    |   movel([0.087836, -1.394012, -2.564950, -0.753428, 1.570796, 1.658633],accel_mss,speed_ms,0,blend_radius_m)
    |   movel([0.088216, -1.393731, -2.565153, -0.753505, 1.570796, 1.659012],accel_mss,speed_ms,0,blend_radius_m)
    |   movel([0.088598, -1.393563, -2.565275, -0.753551, 1.570796, 1.659394],accel_mss,speed_ms,0,blend_radius_m)
    |   movel([0.088951, -1.393516, -2.565308, -0.753564, 1.570796, 1.659747],accel_mss,speed_ms,0,blend_radius_m)
    |   movel([0.089293, -1.393576, -2.565265, -0.753548, 1.570796, 1.660089],accel_mss,speed_ms,0,blend_radius_m)
    |   speed_ms = 0.003
    |   movel([0.089293, -1.380644, -2.559336, -0.772409, 1.570796, 1.660089],accel_mss,speed_ms,0,blend_radius_m)
    |   speed_ms = 1.000
    |   movel([0.089293, -1.355826, -2.547083, -0.809480, 1.570796, 1.660089],accel_mss,speed_ms,0,blend_radius_m)
    |   movel([0.088410, -1.349799, -2.551181, -0.811409, 1.570796, 1.659206],accel_mss,speed_ms,0,blend_radius_m)
    |   movel([0.088410, -1.374726, -2.563511, -0.774153, 1.570796, 1.659206],accel_mss,speed_ms,0,blend_radius_m)
    |   speed_ms = 0.003
    |   movel([0.088410, -1.384438, -2.567999, -0.759952, 1.570796, 1.659206],accel_mss,speed_ms,0,blend_radius_m)
    |   speed_ms = 0.007
    |   movel([0.087081, -1.384926, -2.567651, -0.759811, 1.570796, 1.657878],accel_mss,speed_ms,0,blend_radius_m)
    |   movel([0.085949, -1.385546, -2.567210, -0.759633, 1.570796, 1.656745],accel_mss,speed_ms,0,blend_radius_m)
    |   movel([0.084872, -1.386318, -2.566658, -0.759412, 1.570796, 1.655668],accel_mss,speed_ms,0,blend_radius_m)
    |   movel([0.083929, -1.387193, -2.566033, -0.759163, 1.570796, 1.654725],accel_mss,speed_ms,0,blend_radius_m)
    |   movel([0.083360, -1.387850, -2.565563, -0.758976, 1.570796, 1.654157],accel_mss,speed_ms,0,blend_radius_m)
    |   movel([0.082732, -1.388688, -2.564962, -0.758739, 1.570796, 1.653528],accel_mss,speed_ms,0,blend_radius_m)
    |   movel([0.082181, -1.389503, -2.564376, -0.758510, 1.570796, 1.652978],accel_mss,speed_ms,0,blend_radius_m)
    |   movel([0.081904, -1.390039, -2.563990, -0.758359, 1.570796, 1.652700],accel_mss,speed_ms,0,blend_radius_m)
    |   movel([0.081705, -1.390252, -2.563838, -0.758300, 1.570796, 1.652502],accel_mss,speed_ms,0,blend_radius_m)
    |   movel([0.081566, -1.390049, -2.563984, -0.758357, 1.570796, 1.652362],accel_mss,speed_ms,0,blend_radius_m)
    |   movel([0.081299, -1.389034, -2.564713, -0.758642, 1.570796, 1.652095],accel_mss,speed_ms,0,blend_radius_m)
    |   movel([0.081058, -1.387988, -2.565464, -0.758937, 1.570796, 1.651854],accel_mss,speed_ms,0,blend_radius_m)
    |   movel([0.080915, -1.387123, -2.566083, -0.759183, 1.570796, 1.651712],accel_mss,speed_ms,0,blend_radius_m)
    |   movel([0.080836, -1.386274, -2.566690, -0.759425, 1.570796, 1.651632],accel_mss,speed_ms,0,blend_radius_m)
    |   movel([0.080928, -1.385938, -2.566930, -0.759521, 1.570796, 1.651725],accel_mss,speed_ms,0,blend_radius_m)
    |   movel([0.081186, -1.385742, -2.567070, -0.759577, 1.570796, 1.651983],accel_mss,speed_ms,0,blend_radius_m)
    |   movel([0.081800, -1.385622, -2.567155, -0.759611, 1.570796, 1.652596],accel_mss,speed_ms,0,blend_radius_m)
    |   movel([0.082664, -1.385488, -2.567251, -0.759650, 1.570796, 1.653461],accel_mss,speed_ms,0,blend_radius_m)
    |   movel([0.083900, -1.385238, -2.567429, -0.759721, 1.570796, 1.654697],accel_mss,speed_ms,0,blend_radius_m)
    |   movel([0.085342, -1.384916, -2.567659, -0.759814, 1.570796, 1.656138],accel_mss,speed_ms,0,blend_radius_m)
    |   movel([0.086879, -1.384542, -2.567925, -0.759922, 1.570796, 1.657675],accel_mss,speed_ms,0,blend_radius_m)
    |   movel([0.087796, -1.384317, -2.568085, -0.759987, 1.570796, 1.658593],accel_mss,speed_ms,0,blend_radius_m)
    |   movel([0.088317, -1.384208, -2.568162, -0.760018, 1.570796, 1.659114],accel_mss,speed_ms,0,blend_radius_m)
    |   movel([0.088631, -1.384168, -2.568191, -0.760030, 1.570796, 1.659427],accel_mss,speed_ms,0,blend_radius_m)
    |   movel([0.088410, -1.384438, -2.567999, -0.759952, 1.570796, 1.659206],accel_mss,speed_ms,0,blend_radius_m)
    |   speed_ms = 0.003
    |   movel([0.088410, -1.387720, -2.569479, -0.755191, 1.570796, 1.659206],accel_mss,speed_ms,0,blend_radius_m)
    |   speed_ms = 0.007
    |   movel([0.087081, -1.388207, -2.569130, -0.755052, 1.570796, 1.657878],accel_mss,speed_ms,0,blend_radius_m)
    |   movel([0.085949, -1.388825, -2.568687, -0.754877, 1.570796, 1.656745],accel_mss,speed_ms,0,blend_radius_m)
    |   movel([0.084872, -1.389595, -2.568135, -0.754659, 1.570796, 1.655668],accel_mss,speed_ms,0,blend_radius_m)
    |   movel([0.083929, -1.390467, -2.567508, -0.754414, 1.570796, 1.654725],accel_mss,speed_ms,0,blend_radius_m)
    |   movel([0.083360, -1.391123, -2.567036, -0.754230, 1.570796, 1.654157],accel_mss,speed_ms,0,blend_radius_m)
    |   movel([0.082732, -1.391958, -2.566434, -0.753997, 1.570796, 1.653528],accel_mss,speed_ms,0,blend_radius_m)
    |   movel([0.082181, -1.392771, -2.565848, -0.753771, 1.570796, 1.652978],accel_mss,speed_ms,0,blend_radius_m)
    |   movel([0.081904, -1.393306, -2.565461, -0.753622, 1.570796, 1.652700],accel_mss,speed_ms,0,blend_radius_m)
    |   movel([0.081705, -1.393518, -2.565308, -0.753564, 1.570796, 1.652502],accel_mss,speed_ms,0,blend_radius_m)
    |   movel([0.081566, -1.393315, -2.565454, -0.753620, 1.570796, 1.652362],accel_mss,speed_ms,0,blend_radius_m)
    |   movel([0.081299, -1.392304, -2.566185, -0.753900, 1.570796, 1.652095],accel_mss,speed_ms,0,blend_radius_m)
    |   movel([0.081058, -1.391260, -2.566937, -0.754191, 1.570796, 1.651854],accel_mss,speed_ms,0,blend_radius_m)
    |   movel([0.080915, -1.390398, -2.567558, -0.754433, 1.570796, 1.651712],accel_mss,speed_ms,0,blend_radius_m)
    |   movel([0.080836, -1.389551, -2.568167, -0.754672, 1.570796, 1.651632],accel_mss,speed_ms,0,blend_radius_m)
    |   movel([0.080928, -1.389216, -2.568407, -0.754766, 1.570796, 1.651725],accel_mss,speed_ms,0,blend_radius_m)
    |   movel([0.081186, -1.389020, -2.568547, -0.754822, 1.570796, 1.651983],accel_mss,speed_ms,0,blend_radius_m)
    |   movel([0.081800, -1.388901, -2.568633, -0.754855, 1.570796, 1.652596],accel_mss,speed_ms,0,blend_radius_m)
    |   movel([0.082664, -1.388767, -2.568728, -0.754893, 1.570796, 1.653461],accel_mss,speed_ms,0,blend_radius_m)
    |   movel([0.083900, -1.388518, -2.568907, -0.754964, 1.570796, 1.654697],accel_mss,speed_ms,0,blend_radius_m)
    |   movel([0.085342, -1.388196, -2.569138, -0.755055, 1.570796, 1.656138],accel_mss,speed_ms,0,blend_radius_m)
    |   movel([0.086879, -1.387824, -2.569404, -0.755161, 1.570796, 1.657675],accel_mss,speed_ms,0,blend_radius_m)
    |   movel([0.087796, -1.387599, -2.569565, -0.755225, 1.570796, 1.658593],accel_mss,speed_ms,0,blend_radius_m)
    |   movel([0.088317, -1.387491, -2.569642, -0.755256, 1.570796, 1.659114],accel_mss,speed_ms,0,blend_radius_m)
    |   movel([0.088631, -1.387451, -2.569671, -0.755267, 1.570796, 1.659427],accel_mss,speed_ms,0,blend_radius_m)
    |   movel([0.088410, -1.387720, -2.569479, -0.755191, 1.570796, 1.659206],accel_mss,speed_ms,0,blend_radius_m)
    |   speed_ms = 0.003
    |   movel([0.088410, -1.374726, -2.563511, -0.774153, 1.570796, 1.659206],accel_mss,speed_ms,0,blend_radius_m)
    |   speed_ms = 1.000
    |   movel([0.088410, -1.349799, -2.551181, -0.811409, 1.570796, 1.659206],accel_mss,speed_ms,0,blend_radius_m)
    |   movel([0.072038, -1.358116, -2.545513, -0.808760, 1.570796, 1.642834],accel_mss,speed_ms,0,blend_radius_m)
    |   movel([0.072038, -1.382893, -2.557737, -0.771760, 1.570796, 1.642834],accel_mss,speed_ms,0,blend_radius_m)
    |   speed_ms = 0.003
    |   movel([0.072038, -1.392541, -2.562186, -0.757663, 1.570796, 1.642834],accel_mss,speed_ms,0,blend_radius_m)
    |   speed_ms = 0.007
    |   movel([0.072079, -1.392738, -2.562043, -0.757608, 1.570796, 1.642875],accel_mss,speed_ms,0,blend_radius_m)
    |   movel([0.071854, -1.393010, -2.561846, -0.757533, 1.570796, 1.642650],accel_mss,speed_ms,0,blend_radius_m)
    |   movel([0.071545, -1.393082, -2.561794, -0.757513, 1.570796, 1.642341],accel_mss,speed_ms,0,blend_radius_m)
    |   movel([0.071303, -1.393090, -2.561788, -0.757511, 1.570796, 1.642100],accel_mss,speed_ms,0,blend_radius_m)
    |   movel([0.071035, -1.393108, -2.561775, -0.757506, 1.570796, 1.641831],accel_mss,speed_ms,0,blend_radius_m)
    |   movel([0.070605, -1.393174, -2.561727, -0.757488, 1.570796, 1.641402],accel_mss,speed_ms,0,blend_radius_m)
    |   movel([0.070116, -1.393271, -2.561657, -0.757461, 1.570796, 1.640912],accel_mss,speed_ms,0,blend_radius_m)
    |   movel([0.069632, -1.393385, -2.561575, -0.757430, 1.570796, 1.640429],accel_mss,speed_ms,0,blend_radius_m)
    |   movel([0.068674, -1.393599, -2.561419, -0.757371, 1.570796, 1.639470],accel_mss,speed_ms,0,blend_radius_m)
    |   movel([0.068254, -1.393580, -2.561433, -0.757376, 1.570796, 1.639050],accel_mss,speed_ms,0,blend_radius_m)
    |   movel([0.068198, -1.393373, -2.561583, -0.757433, 1.570796, 1.638995],accel_mss,speed_ms,0,blend_radius_m)
    |   movel([0.068476, -1.392973, -2.561872, -0.757543, 1.570796, 1.639272],accel_mss,speed_ms,0,blend_radius_m)
    |   movel([0.068846, -1.392690, -2.562077, -0.757621, 1.570796, 1.639642],accel_mss,speed_ms,0,blend_radius_m)
    |   movel([0.069096, -1.392605, -2.562139, -0.757645, 1.570796, 1.639893],accel_mss,speed_ms,0,blend_radius_m)
    |   movel([0.069570, -1.392494, -2.562220, -0.757676, 1.570796, 1.640367],accel_mss,speed_ms,0,blend_radius_m)
    |   movel([0.070403, -1.392329, -2.562339, -0.757721, 1.570796, 1.641200],accel_mss,speed_ms,0,blend_radius_m)
    |   movel([0.071125, -1.392221, -2.562417, -0.757751, 1.570796, 1.641922],accel_mss,speed_ms,0,blend_radius_m)
    |   movel([0.071701, -1.392164, -2.562458, -0.757767, 1.570796, 1.642497],accel_mss,speed_ms,0,blend_radius_m)
    |   movel([0.071942, -1.392284, -2.562371, -0.757734, 1.570796, 1.642738],accel_mss,speed_ms,0,blend_radius_m)
    |   movel([0.072038, -1.392541, -2.562186, -0.757663, 1.570796, 1.642834],accel_mss,speed_ms,0,blend_radius_m)
    |   speed_ms = 0.003
    |   movel([0.072038, -1.395800, -2.563652, -0.752937, 1.570796, 1.642834],accel_mss,speed_ms,0,blend_radius_m)
    |   speed_ms = 0.007
    |   movel([0.072079, -1.395997, -2.563509, -0.752883, 1.570796, 1.642875],accel_mss,speed_ms,0,blend_radius_m)
    |   movel([0.071854, -1.396269, -2.563311, -0.752809, 1.570796, 1.642650],accel_mss,speed_ms,0,blend_radius_m)
    |   movel([0.071545, -1.396340, -2.563259, -0.752790, 1.570796, 1.642341],accel_mss,speed_ms,0,blend_radius_m)
    |   movel([0.071303, -1.396348, -2.563254, -0.752788, 1.570796, 1.642100],accel_mss,speed_ms,0,blend_radius_m)
    |   movel([0.071035, -1.396366, -2.563240, -0.752783, 1.570796, 1.641831],accel_mss,speed_ms,0,blend_radius_m)
    |   movel([0.070605, -1.396432, -2.563192, -0.752765, 1.570796, 1.641402],accel_mss,speed_ms,0,blend_radius_m)
    |   movel([0.070116, -1.396529, -2.563122, -0.752738, 1.570796, 1.640912],accel_mss,speed_ms,0,blend_radius_m)
    |   movel([0.069632, -1.396642, -2.563039, -0.752708, 1.570796, 1.640429],accel_mss,speed_ms,0,blend_radius_m)
    |   movel([0.068674, -1.396856, -2.562883, -0.752649, 1.570796, 1.639470],accel_mss,speed_ms,0,blend_radius_m)
    |   movel([0.068254, -1.396836, -2.562898, -0.752655, 1.570796, 1.639050],accel_mss,speed_ms,0,blend_radius_m)
    |   movel([0.068198, -1.396630, -2.563048, -0.752711, 1.570796, 1.638995],accel_mss,speed_ms,0,blend_radius_m)
    |   movel([0.068476, -1.396232, -2.563338, -0.752819, 1.570796, 1.639272],accel_mss,speed_ms,0,blend_radius_m)
    |   movel([0.068846, -1.395949, -2.563543, -0.752896, 1.570796, 1.639642],accel_mss,speed_ms,0,blend_radius_m)
    |   movel([0.069096, -1.395864, -2.563605, -0.752919, 1.570796, 1.639893],accel_mss,speed_ms,0,blend_radius_m)
    |   movel([0.069570, -1.395754, -2.563686, -0.752950, 1.570796, 1.640367],accel_mss,speed_ms,0,blend_radius_m)
    |   movel([0.070403, -1.395589, -2.563805, -0.752995, 1.570796, 1.641200],accel_mss,speed_ms,0,blend_radius_m)
    |   movel([0.071125, -1.395481, -2.563884, -0.753024, 1.570796, 1.641922],accel_mss,speed_ms,0,blend_radius_m)
    |   movel([0.071701, -1.395425, -2.563925, -0.753040, 1.570796, 1.642497],accel_mss,speed_ms,0,blend_radius_m)
    |   movel([0.071942, -1.395544, -2.563838, -0.753007, 1.570796, 1.642738],accel_mss,speed_ms,0,blend_radius_m)
    |   movel([0.072038, -1.395800, -2.563652, -0.752937, 1.570796, 1.642834],accel_mss,speed_ms,0,blend_radius_m)
    |   speed_ms = 0.003
    |   movel([0.072038, -1.382893, -2.557737, -0.771760, 1.570796, 1.642834],accel_mss,speed_ms,0,blend_radius_m)
    |   speed_ms = 1.000
    |   movel([0.072038, -1.358116, -2.545513, -0.808760, 1.570796, 1.642834],accel_mss,speed_ms,0,blend_radius_m)
    |   movel([0.071087, -1.359327, -2.544680, -0.808382, 1.570796, 1.641883],accel_mss,speed_ms,0,blend_radius_m)
    |   movel([0.071087, -1.384082, -2.556888, -0.771419, 1.570796, 1.641883],accel_mss,speed_ms,0,blend_radius_m)
    |   speed_ms = 0.003
    |   movel([0.071087, -1.393720, -2.561331, -0.757337, 1.570796, 1.641883],accel_mss,speed_ms,0,blend_radius_m)
    |   speed_ms = 0.007
    |   movel([0.071759, -1.393816, -2.561262, -0.757311, 1.570796, 1.642556],accel_mss,speed_ms,0,blend_radius_m)
    |   movel([0.071953, -1.393945, -2.561168, -0.757276, 1.570796, 1.642749],accel_mss,speed_ms,0,blend_radius_m)
    |   movel([0.072032, -1.394114, -2.561046, -0.757229, 1.570796, 1.642829],accel_mss,speed_ms,0,blend_radius_m)
    |   movel([0.071840, -1.394423, -2.560821, -0.757144, 1.570796, 1.642637],accel_mss,speed_ms,0,blend_radius_m)
    |   movel([0.071514, -1.394499, -2.560766, -0.757124, 1.570796, 1.642311],accel_mss,speed_ms,0,blend_radius_m)
    |   movel([0.071242, -1.394533, -2.560742, -0.757114, 1.570796, 1.642039],accel_mss,speed_ms,0,blend_radius_m)
    |   movel([0.070950, -1.394556, -2.560725, -0.757108, 1.570796, 1.641746],accel_mss,speed_ms,0,blend_radius_m)
    |   movel([0.070596, -1.394590, -2.560700, -0.757099, 1.570796, 1.641393],accel_mss,speed_ms,0,blend_radius_m)
    |   movel([0.070127, -1.394658, -2.560651, -0.757080, 1.570796, 1.640923],accel_mss,speed_ms,0,blend_radius_m)
    |   movel([0.069629, -1.394746, -2.560587, -0.757056, 1.570796, 1.640426],accel_mss,speed_ms,0,blend_radius_m)
    |   movel([0.069177, -1.394842, -2.560517, -0.757030, 1.570796, 1.639973],accel_mss,speed_ms,0,blend_radius_m)
    |   movel([0.068658, -1.394956, -2.560434, -0.756999, 1.570796, 1.639454],accel_mss,speed_ms,0,blend_radius_m)
    |   movel([0.068335, -1.395002, -2.560401, -0.756986, 1.570796, 1.639131],accel_mss,speed_ms,0,blend_radius_m)
    |   movel([0.068017, -1.394943, -2.560443, -0.757002, 1.570796, 1.638813],accel_mss,speed_ms,0,blend_radius_m)
    |   movel([0.068021, -1.394682, -2.560633, -0.757074, 1.570796, 1.638818],accel_mss,speed_ms,0,blend_radius_m)
    |   movel([0.068685, -1.394201, -2.560983, -0.757205, 1.570796, 1.639482],accel_mss,speed_ms,0,blend_radius_m)
    |   movel([0.069886, -1.393897, -2.561203, -0.757289, 1.570796, 1.640683],accel_mss,speed_ms,0,blend_radius_m)
    |   movel([0.071087, -1.393720, -2.561331, -0.757337, 1.570796, 1.641883],accel_mss,speed_ms,0,blend_radius_m)
    |   speed_ms = 0.003
    |   movel([0.071087, -1.396977, -2.562796, -0.752617, 1.570796, 1.641883],accel_mss,speed_ms,0,blend_radius_m)
    |   speed_ms = 0.007
    |   movel([0.071759, -1.397072, -2.562726, -0.752591, 1.570796, 1.642556],accel_mss,speed_ms,0,blend_radius_m)
    |   movel([0.071953, -1.397201, -2.562632, -0.752556, 1.570796, 1.642749],accel_mss,speed_ms,0,blend_radius_m)
    |   movel([0.072032, -1.397369, -2.562509, -0.752510, 1.570796, 1.642829],accel_mss,speed_ms,0,blend_radius_m)
    |   movel([0.071840, -1.397678, -2.562284, -0.752427, 1.570796, 1.642637],accel_mss,speed_ms,0,blend_radius_m)
    |   movel([0.071514, -1.397753, -2.562229, -0.752406, 1.570796, 1.642311],accel_mss,speed_ms,0,blend_radius_m)
    |   movel([0.071242, -1.397787, -2.562205, -0.752397, 1.570796, 1.642039],accel_mss,speed_ms,0,blend_radius_m)
    |   movel([0.070950, -1.397810, -2.562188, -0.752391, 1.570796, 1.641746],accel_mss,speed_ms,0,blend_radius_m)
    |   movel([0.070596, -1.397844, -2.562163, -0.752382, 1.570796, 1.641393],accel_mss,speed_ms,0,blend_radius_m)
    |   movel([0.070127, -1.397911, -2.562114, -0.752364, 1.570796, 1.640923],accel_mss,speed_ms,0,blend_radius_m)
    |   movel([0.069629, -1.398000, -2.562049, -0.752340, 1.570796, 1.640426],accel_mss,speed_ms,0,blend_radius_m)
    |   movel([0.069177, -1.398096, -2.561979, -0.752314, 1.570796, 1.639973],accel_mss,speed_ms,0,blend_radius_m)
    |   movel([0.068658, -1.398209, -2.561896, -0.752283, 1.570796, 1.639454],accel_mss,speed_ms,0,blend_radius_m)
    |   movel([0.068335, -1.398255, -2.561863, -0.752271, 1.570796, 1.639131],accel_mss,speed_ms,0,blend_radius_m)
    |   movel([0.068017, -1.398196, -2.561906, -0.752287, 1.570796, 1.638813],accel_mss,speed_ms,0,blend_radius_m)
    |   movel([0.068021, -1.397936, -2.562096, -0.752357, 1.570796, 1.638818],accel_mss,speed_ms,0,blend_radius_m)
    |   movel([0.068685, -1.397456, -2.562446, -0.752487, 1.570796, 1.639482],accel_mss,speed_ms,0,blend_radius_m)
    |   movel([0.069886, -1.397153, -2.562667, -0.752569, 1.570796, 1.640683],accel_mss,speed_ms,0,blend_radius_m)
    |   movel([0.071087, -1.396977, -2.562796, -0.752617, 1.570796, 1.641883],accel_mss,speed_ms,0,blend_radius_m)
    |   speed_ms = 0.003
    |   movel([0.071087, -1.384082, -2.556888, -0.771419, 1.570796, 1.641883],accel_mss,speed_ms,0,blend_radius_m)
    |   speed_ms = 1.000
    |   movel([0.071087, -1.359327, -2.544680, -0.808382, 1.570796, 1.641883],accel_mss,speed_ms,0,blend_radius_m)
    |   movel([0.070689, -1.360858, -2.543624, -0.807908, 1.570796, 1.641485],accel_mss,speed_ms,0,blend_radius_m)
    |   movel([0.070689, -1.385584, -2.555813, -0.770992, 1.570796, 1.641485],accel_mss,speed_ms,0,blend_radius_m)
    |   speed_ms = 0.003
    |   movel([0.070689, -1.395211, -2.560249, -0.756929, 1.570796, 1.641485],accel_mss,speed_ms,0,blend_radius_m)
    |   speed_ms = 0.007
    |   movel([0.071288, -1.395336, -2.560158, -0.756895, 1.570796, 1.642084],accel_mss,speed_ms,0,blend_radius_m)
    |   movel([0.071443, -1.395487, -2.560048, -0.756854, 1.570796, 1.642240],accel_mss,speed_ms,0,blend_radius_m)
    |   movel([0.071331, -1.395822, -2.559804, -0.756763, 1.570796, 1.642128],accel_mss,speed_ms,0,blend_radius_m)
    |   movel([0.070938, -1.395963, -2.559701, -0.756724, 1.570796, 1.641734],accel_mss,speed_ms,0,blend_radius_m)
    |   movel([0.070676, -1.396000, -2.559674, -0.756714, 1.570796, 1.641472],accel_mss,speed_ms,0,blend_radius_m)
    |   movel([0.070376, -1.396032, -2.559651, -0.756706, 1.570796, 1.641172],accel_mss,speed_ms,0,blend_radius_m)
    |   movel([0.070079, -1.396055, -2.559635, -0.756699, 1.570796, 1.640875],accel_mss,speed_ms,0,blend_radius_m)
    |   movel([0.069755, -1.396088, -2.559611, -0.756691, 1.570796, 1.640551],accel_mss,speed_ms,0,blend_radius_m)
    |   movel([0.069368, -1.396148, -2.559567, -0.756674, 1.570796, 1.640165],accel_mss,speed_ms,0,blend_radius_m)
    |   movel([0.068988, -1.396224, -2.559511, -0.756654, 1.570796, 1.639784],accel_mss,speed_ms,0,blend_radius_m)
    |   movel([0.068671, -1.396306, -2.559452, -0.756631, 1.570796, 1.639468],accel_mss,speed_ms,0,blend_radius_m)
    |   movel([0.068109, -1.396441, -2.559353, -0.756595, 1.570796, 1.638905],accel_mss,speed_ms,0,blend_radius_m)
    |   movel([0.067804, -1.396414, -2.559373, -0.756602, 1.570796, 1.638600],accel_mss,speed_ms,0,blend_radius_m)
    |   movel([0.067930, -1.395974, -2.559694, -0.756722, 1.570796, 1.638726],accel_mss,speed_ms,0,blend_radius_m)
    |   movel([0.068477, -1.395624, -2.559948, -0.756817, 1.570796, 1.639273],accel_mss,speed_ms,0,blend_radius_m)
    |   movel([0.069587, -1.395350, -2.560147, -0.756891, 1.570796, 1.640383],accel_mss,speed_ms,0,blend_radius_m)
    |   movel([0.070689, -1.395211, -2.560249, -0.756929, 1.570796, 1.641485],accel_mss,speed_ms,0,blend_radius_m)
    |   speed_ms = 0.003
    |   movel([0.070689, -1.398463, -2.561711, -0.752215, 1.570796, 1.641485],accel_mss,speed_ms,0,blend_radius_m)
    |   speed_ms = 0.007
    |   movel([0.071288, -1.398588, -2.561619, -0.752182, 1.570796, 1.642084],accel_mss,speed_ms,0,blend_radius_m)
    |   movel([0.071443, -1.398738, -2.561510, -0.752141, 1.570796, 1.642240],accel_mss,speed_ms,0,blend_radius_m)
    |   movel([0.071331, -1.399073, -2.561265, -0.752051, 1.570796, 1.642128],accel_mss,speed_ms,0,blend_radius_m)
    |   movel([0.070938, -1.399214, -2.561162, -0.752014, 1.570796, 1.641734],accel_mss,speed_ms,0,blend_radius_m)
    |   movel([0.070676, -1.399250, -2.561135, -0.752004, 1.570796, 1.641472],accel_mss,speed_ms,0,blend_radius_m)
    |   movel([0.070376, -1.399282, -2.561112, -0.751995, 1.570796, 1.641172],accel_mss,speed_ms,0,blend_radius_m)
    |   movel([0.070079, -1.399305, -2.561095, -0.751989, 1.570796, 1.640875],accel_mss,speed_ms,0,blend_radius_m)
    |   movel([0.069755, -1.399338, -2.561071, -0.751980, 1.570796, 1.640551],accel_mss,speed_ms,0,blend_radius_m)
    |   movel([0.069368, -1.399397, -2.561027, -0.751964, 1.570796, 1.640165],accel_mss,speed_ms,0,blend_radius_m)
    |   movel([0.068988, -1.399473, -2.560972, -0.751944, 1.570796, 1.639784],accel_mss,speed_ms,0,blend_radius_m)
    |   movel([0.068671, -1.399555, -2.560912, -0.751922, 1.570796, 1.639468],accel_mss,speed_ms,0,blend_radius_m)
    |   movel([0.068109, -1.399690, -2.560813, -0.751886, 1.570796, 1.638905],accel_mss,speed_ms,0,blend_radius_m)
    |   movel([0.067804, -1.399663, -2.560833, -0.751893, 1.570796, 1.638600],accel_mss,speed_ms,0,blend_radius_m)
    |   movel([0.067930, -1.399224, -2.561154, -0.752011, 1.570796, 1.638726],accel_mss,speed_ms,0,blend_radius_m)
    |   movel([0.068477, -1.398875, -2.561409, -0.752104, 1.570796, 1.639273],accel_mss,speed_ms,0,blend_radius_m)
    |   movel([0.069587, -1.398602, -2.561609, -0.752178, 1.570796, 1.640383],accel_mss,speed_ms,0,blend_radius_m)
    |   movel([0.070689, -1.398463, -2.561711, -0.752215, 1.570796, 1.641485],accel_mss,speed_ms,0,blend_radius_m)
    |   speed_ms = 0.003
    |   movel([0.070689, -1.385584, -2.555813, -0.770992, 1.570796, 1.641485],accel_mss,speed_ms,0,blend_radius_m)
    |   speed_ms = 1.000
    |   movel([0.070689, -1.360858, -2.543624, -0.807908, 1.570796, 1.641485],accel_mss,speed_ms,0,blend_radius_m)
    |   movel([0.069782, -1.362641, -2.542390, -0.807359, 1.570796, 1.640579],accel_mss,speed_ms,0,blend_radius_m)
    |   movel([0.069782, -1.387335, -2.554556, -0.770498, 1.570796, 1.640579],accel_mss,speed_ms,0,blend_radius_m)
    |   speed_ms = 0.003
    |   movel([0.069782, -1.396948, -2.558984, -0.756458, 1.570796, 1.640579],accel_mss,speed_ms,0,blend_radius_m)
    |   speed_ms = 0.007
    |   movel([0.070081, -1.397018, -2.558932, -0.756439, 1.570796, 1.640877],accel_mss,speed_ms,0,blend_radius_m)
    |   movel([0.070082, -1.397273, -2.558746, -0.756370, 1.570796, 1.640878],accel_mss,speed_ms,0,blend_radius_m)
    |   movel([0.069829, -1.397430, -2.558632, -0.756328, 1.570796, 1.640625],accel_mss,speed_ms,0,blend_radius_m)
    |   movel([0.069576, -1.397509, -2.558574, -0.756306, 1.570796, 1.640372],accel_mss,speed_ms,0,blend_radius_m)
    |   movel([0.069100, -1.397609, -2.558501, -0.756279, 1.570796, 1.639897],accel_mss,speed_ms,0,blend_radius_m)
    |   movel([0.068697, -1.397625, -2.558489, -0.756275, 1.570796, 1.639493],accel_mss,speed_ms,0,blend_radius_m)
    |   movel([0.068424, -1.397557, -2.558538, -0.756293, 1.570796, 1.639220],accel_mss,speed_ms,0,blend_radius_m)
    |   movel([0.068377, -1.397306, -2.558722, -0.756361, 1.570796, 1.639174],accel_mss,speed_ms,0,blend_radius_m)
    |   movel([0.068857, -1.397068, -2.558896, -0.756425, 1.570796, 1.639653],accel_mss,speed_ms,0,blend_radius_m)
    |   movel([0.069345, -1.396961, -2.558974, -0.756454, 1.570796, 1.640141],accel_mss,speed_ms,0,blend_radius_m)
    |   movel([0.069782, -1.396948, -2.558984, -0.756458, 1.570796, 1.640579],accel_mss,speed_ms,0,blend_radius_m)
    |   speed_ms = 0.003
    |   movel([0.069782, -1.400195, -2.560443, -0.751751, 1.570796, 1.640579],accel_mss,speed_ms,0,blend_radius_m)
    |   speed_ms = 0.007
    |   movel([0.070081, -1.400265, -2.560391, -0.751733, 1.570796, 1.640877],accel_mss,speed_ms,0,blend_radius_m)
    |   movel([0.070082, -1.400520, -2.560205, -0.751665, 1.570796, 1.640878],accel_mss,speed_ms,0,blend_radius_m)
    |   movel([0.069829, -1.400676, -2.560090, -0.751623, 1.570796, 1.640625],accel_mss,speed_ms,0,blend_radius_m)
    |   movel([0.069576, -1.400755, -2.560032, -0.751602, 1.570796, 1.640372],accel_mss,speed_ms,0,blend_radius_m)
    |   movel([0.069100, -1.400855, -2.559959, -0.751576, 1.570796, 1.639897],accel_mss,speed_ms,0,blend_radius_m)
    |   movel([0.068697, -1.400871, -2.559947, -0.751571, 1.570796, 1.639493],accel_mss,speed_ms,0,blend_radius_m)
    |   movel([0.068424, -1.400803, -2.559996, -0.751589, 1.570796, 1.639220],accel_mss,speed_ms,0,blend_radius_m)
    |   movel([0.068377, -1.400553, -2.560180, -0.751656, 1.570796, 1.639174],accel_mss,speed_ms,0,blend_radius_m)
    |   movel([0.068857, -1.400315, -2.560355, -0.751719, 1.570796, 1.639653],accel_mss,speed_ms,0,blend_radius_m)
    |   movel([0.069345, -1.400209, -2.560433, -0.751748, 1.570796, 1.640141],accel_mss,speed_ms,0,blend_radius_m)
    |   movel([0.069782, -1.400195, -2.560443, -0.751751, 1.570796, 1.640579],accel_mss,speed_ms,0,blend_radius_m)
    |   speed_ms = 0.003
    |   movel([0.069782, -1.387335, -2.554556, -0.770498, 1.570796, 1.640579],accel_mss,speed_ms,0,blend_radius_m)
    |   speed_ms = 1.000
    |   movel([0.069782, -1.362641, -2.542390, -0.807359, 1.570796, 1.640579],accel_mss,speed_ms,0,blend_radius_m)
    |   movel([0.070729, -1.364236, -2.541282, -0.806871, 1.570796, 1.641526],accel_mss,speed_ms,0,blend_radius_m)
    |   movel([0.070729, -1.388900, -2.553429, -0.770060, 1.570796, 1.641526],accel_mss,speed_ms,0,blend_radius_m)
    |   speed_ms = 0.003
    |   movel([0.070729, -1.398501, -2.557849, -0.756040, 1.570796, 1.641526],accel_mss,speed_ms,0,blend_radius_m)
    |   speed_ms = 0.007
    |   movel([0.071066, -1.398674, -2.557722, -0.755993, 1.570796, 1.641863],accel_mss,speed_ms,0,blend_radius_m)
    |   movel([0.071301, -1.399152, -2.557371, -0.755865, 1.570796, 1.642097],accel_mss,speed_ms,0,blend_radius_m)
    |   movel([0.071374, -1.399599, -2.557044, -0.755746, 1.570796, 1.642170],accel_mss,speed_ms,0,blend_radius_m)
    |   movel([0.071289, -1.400063, -2.556703, -0.755623, 1.570796, 1.642086],accel_mss,speed_ms,0,blend_radius_m)
    |   movel([0.071044, -1.400592, -2.556314, -0.755483, 1.570796, 1.641841],accel_mss,speed_ms,0,blend_radius_m)
    |   movel([0.070729, -1.401057, -2.555973, -0.755360, 1.570796, 1.641525],accel_mss,speed_ms,0,blend_radius_m)
    |   movel([0.070393, -1.401405, -2.555716, -0.755268, 1.570796, 1.641189],accel_mss,speed_ms,0,blend_radius_m)
    |   movel([0.069983, -1.401684, -2.555511, -0.755194, 1.570796, 1.640780],accel_mss,speed_ms,0,blend_radius_m)
    |   movel([0.069443, -1.401936, -2.555325, -0.755128, 1.570796, 1.640239],accel_mss,speed_ms,0,blend_radius_m)
    |   movel([0.069084, -1.402074, -2.555223, -0.755091, 1.570796, 1.639880],accel_mss,speed_ms,0,blend_radius_m)
    |   movel([0.068795, -1.402105, -2.555201, -0.755083, 1.570796, 1.639592],accel_mss,speed_ms,0,blend_radius_m)
    |   movel([0.068720, -1.401890, -2.555359, -0.755140, 1.570796, 1.639516],accel_mss,speed_ms,0,blend_radius_m)
    |   movel([0.069417, -1.401321, -2.555778, -0.755290, 1.570796, 1.640213],accel_mss,speed_ms,0,blend_radius_m)
    |   movel([0.069950, -1.400675, -2.556253, -0.755461, 1.570796, 1.640746],accel_mss,speed_ms,0,blend_radius_m)
    |   movel([0.070338, -1.399931, -2.556800, -0.755658, 1.570796, 1.641134],accel_mss,speed_ms,0,blend_radius_m)
    |   movel([0.070527, -1.399177, -2.557353, -0.755859, 1.570796, 1.641323],accel_mss,speed_ms,0,blend_radius_m)
    |   movel([0.070602, -1.398709, -2.557696, -0.755984, 1.570796, 1.641398],accel_mss,speed_ms,0,blend_radius_m)
    |   speed_ms = 0.003
    |   movel([0.070729, -1.401744, -2.559305, -0.751340, 1.570796, 1.641526],accel_mss,speed_ms,0,blend_radius_m)
    |   speed_ms = 0.007
    |   movel([0.071066, -1.401917, -2.559178, -0.751295, 1.570796, 1.641863],accel_mss,speed_ms,0,blend_radius_m)
    |   movel([0.071301, -1.402394, -2.558827, -0.751169, 1.570796, 1.642097],accel_mss,speed_ms,0,blend_radius_m)
    |   movel([0.071374, -1.402839, -2.558498, -0.751052, 1.570796, 1.642170],accel_mss,speed_ms,0,blend_radius_m)
    |   movel([0.071289, -1.403302, -2.558157, -0.750930, 1.570796, 1.642086],accel_mss,speed_ms,0,blend_radius_m)
    |   movel([0.071044, -1.403829, -2.557767, -0.750792, 1.570796, 1.641841],accel_mss,speed_ms,0,blend_radius_m)
    |   movel([0.070729, -1.404292, -2.557425, -0.750671, 1.570796, 1.641525],accel_mss,speed_ms,0,blend_radius_m)
    |   movel([0.070393, -1.404640, -2.557168, -0.750581, 1.570796, 1.641189],accel_mss,speed_ms,0,blend_radius_m)
    |   movel([0.069983, -1.404918, -2.556962, -0.750509, 1.570796, 1.640780],accel_mss,speed_ms,0,blend_radius_m)
    |   movel([0.069443, -1.405170, -2.556776, -0.750444, 1.570796, 1.640239],accel_mss,speed_ms,0,blend_radius_m)
    |   movel([0.069084, -1.405308, -2.556674, -0.750408, 1.570796, 1.639880],accel_mss,speed_ms,0,blend_radius_m)
    |   movel([0.068795, -1.405338, -2.556651, -0.750400, 1.570796, 1.639592],accel_mss,speed_ms,0,blend_radius_m)
    |   movel([0.068720, -1.405124, -2.556810, -0.750455, 1.570796, 1.639516],accel_mss,speed_ms,0,blend_radius_m)
    |   movel([0.069417, -1.404556, -2.557230, -0.750603, 1.570796, 1.640213],accel_mss,speed_ms,0,blend_radius_m)
    |   movel([0.069950, -1.403912, -2.557706, -0.750771, 1.570796, 1.640746],accel_mss,speed_ms,0,blend_radius_m)
    |   movel([0.070338, -1.403170, -2.558255, -0.750965, 1.570796, 1.641134],accel_mss,speed_ms,0,blend_radius_m)
    |   movel([0.070527, -1.402418, -2.558808, -0.751162, 1.570796, 1.641323],accel_mss,speed_ms,0,blend_radius_m)
    |   movel([0.070602, -1.401952, -2.559152, -0.751285, 1.570796, 1.641398],accel_mss,speed_ms,0,blend_radius_m)
    |   speed_ms = 0.003
    |   movel([0.070729, -1.388900, -2.553429, -0.770060, 1.570796, 1.641526],accel_mss,speed_ms,0,blend_radius_m)
    |   speed_ms = 1.000
    |   movel([0.070729, -1.364236, -2.541282, -0.806871, 1.570796, 1.641526],accel_mss,speed_ms,0,blend_radius_m)
    |   movel([0.067029, -1.364169, -2.541328, -0.806891, 1.570796, 1.637826],accel_mss,speed_ms,0,blend_radius_m)
    |   movel([0.067029, -1.388835, -2.553476, -0.770078, 1.570796, 1.637826],accel_mss,speed_ms,0,blend_radius_m)
    |   speed_ms = 0.003
    |   movel([0.067029, -1.398436, -2.557896, -0.756057, 1.570796, 1.637826],accel_mss,speed_ms,0,blend_radius_m)
    |   speed_ms = 0.007
    |   movel([0.066484, -1.399101, -2.557408, -0.755879, 1.570796, 1.637280],accel_mss,speed_ms,0,blend_radius_m)
    |   movel([0.066042, -1.399666, -2.556994, -0.755728, 1.570796, 1.636839],accel_mss,speed_ms,0,blend_radius_m)
    |   movel([0.065758, -1.400184, -2.556614, -0.755591, 1.570796, 1.636554],accel_mss,speed_ms,0,blend_radius_m)
    |   movel([0.065615, -1.400700, -2.556235, -0.755454, 1.570796, 1.636412],accel_mss,speed_ms,0,blend_radius_m)
    |   movel([0.065596, -1.401254, -2.555828, -0.755308, 1.570796, 1.636393],accel_mss,speed_ms,0,blend_radius_m)
    |   movel([0.065612, -1.401543, -2.555615, -0.755231, 1.570796, 1.636409],accel_mss,speed_ms,0,blend_radius_m)
    |   movel([0.065467, -1.401787, -2.555435, -0.755167, 1.570796, 1.636263],accel_mss,speed_ms,0,blend_radius_m)
    |   movel([0.065143, -1.401626, -2.555553, -0.755209, 1.570796, 1.635939],accel_mss,speed_ms,0,blend_radius_m)
    |   movel([0.064965, -1.401144, -2.555908, -0.755337, 1.570796, 1.635761],accel_mss,speed_ms,0,blend_radius_m)
    |   movel([0.064953, -1.400540, -2.556352, -0.755496, 1.570796, 1.635750],accel_mss,speed_ms,0,blend_radius_m)
    |   movel([0.065148, -1.399997, -2.556752, -0.755640, 1.570796, 1.635945],accel_mss,speed_ms,0,blend_radius_m)
    |   movel([0.065500, -1.399499, -2.557117, -0.755773, 1.570796, 1.636296],accel_mss,speed_ms,0,blend_radius_m)
    |   movel([0.065982, -1.398991, -2.557490, -0.755909, 1.570796, 1.636779],accel_mss,speed_ms,0,blend_radius_m)
    |   movel([0.066487, -1.398571, -2.557797, -0.756021, 1.570796, 1.637283],accel_mss,speed_ms,0,blend_radius_m)
    |   movel([0.066886, -1.398369, -2.557945, -0.756075, 1.570796, 1.637682],accel_mss,speed_ms,0,blend_radius_m)
    |   speed_ms = 0.003
    |   movel([0.067029, -1.401679, -2.559353, -0.751357, 1.570796, 1.637826],accel_mss,speed_ms,0,blend_radius_m)
    |   speed_ms = 0.007
    |   movel([0.066484, -1.402343, -2.558864, -0.751182, 1.570796, 1.637280],accel_mss,speed_ms,0,blend_radius_m)
    |   movel([0.066042, -1.402906, -2.558449, -0.751034, 1.570796, 1.636839],accel_mss,speed_ms,0,blend_radius_m)
    |   movel([0.065758, -1.403423, -2.558068, -0.750899, 1.570796, 1.636554],accel_mss,speed_ms,0,blend_radius_m)
    |   movel([0.065615, -1.403937, -2.557688, -0.750764, 1.570796, 1.636412],accel_mss,speed_ms,0,blend_radius_m)
    |   movel([0.065596, -1.404489, -2.557280, -0.750620, 1.570796, 1.636393],accel_mss,speed_ms,0,blend_radius_m)
    |   movel([0.065612, -1.404777, -2.557066, -0.750545, 1.570796, 1.636409],accel_mss,speed_ms,0,blend_radius_m)
    |   movel([0.065467, -1.405021, -2.556886, -0.750482, 1.570796, 1.636263],accel_mss,speed_ms,0,blend_radius_m)
    |   movel([0.065143, -1.404861, -2.557005, -0.750524, 1.570796, 1.635939],accel_mss,speed_ms,0,blend_radius_m)
    |   movel([0.064965, -1.404380, -2.557361, -0.750649, 1.570796, 1.635761],accel_mss,speed_ms,0,blend_radius_m)
    |   movel([0.064953, -1.403778, -2.557805, -0.750806, 1.570796, 1.635750],accel_mss,speed_ms,0,blend_radius_m)
    |   movel([0.065148, -1.403236, -2.558206, -0.750948, 1.570796, 1.635945],accel_mss,speed_ms,0,blend_radius_m)
    |   movel([0.065500, -1.402739, -2.558572, -0.751078, 1.570796, 1.636296],accel_mss,speed_ms,0,blend_radius_m)
    |   movel([0.065982, -1.402232, -2.558945, -0.751211, 1.570796, 1.636779],accel_mss,speed_ms,0,blend_radius_m)
    |   movel([0.066487, -1.401814, -2.559253, -0.751322, 1.570796, 1.637283],accel_mss,speed_ms,0,blend_radius_m)
    |   movel([0.066886, -1.401612, -2.559402, -0.751375, 1.570796, 1.637682],accel_mss,speed_ms,0,blend_radius_m)
    |   speed_ms = 0.003
    |   movel([0.067029, -1.388835, -2.553476, -0.770078, 1.570796, 1.637826],accel_mss,speed_ms,0,blend_radius_m)
    |   speed_ms = 1.000
    |   movel([0.067029, -1.364169, -2.541328, -0.806891, 1.570796, 1.637826],accel_mss,speed_ms,0,blend_radius_m)
    |   movel([0.063503, -1.363293, -2.541937, -0.807159, 1.570796, 1.634299],accel_mss,speed_ms,0,blend_radius_m)
    |   movel([0.063503, -1.387975, -2.554096, -0.770318, 1.570796, 1.634299],accel_mss,speed_ms,0,blend_radius_m)
    |   speed_ms = 0.003
    |   movel([0.063503, -1.397583, -2.558520, -0.756286, 1.570796, 1.634299],accel_mss,speed_ms,0,blend_radius_m)
    |   speed_ms = 0.007
    |   movel([0.062657, -1.398693, -2.557707, -0.755988, 1.570796, 1.633454],accel_mss,speed_ms,0,blend_radius_m)
    |   movel([0.061791, -1.399822, -2.556880, -0.755687, 1.570796, 1.632587],accel_mss,speed_ms,0,blend_radius_m)
    |   movel([0.061009, -1.400829, -2.556140, -0.755420, 1.570796, 1.631805],accel_mss,speed_ms,0,blend_radius_m)
    |   movel([0.060348, -1.401674, -2.555518, -0.755197, 1.570796, 1.631144],accel_mss,speed_ms,0,blend_radius_m)
    |   movel([0.060139, -1.401920, -2.555337, -0.755132, 1.570796, 1.630935],accel_mss,speed_ms,0,blend_radius_m)
    |   movel([0.059822, -1.402269, -2.555080, -0.755041, 1.570796, 1.630619],accel_mss,speed_ms,0,blend_radius_m)
    |   movel([0.059929, -1.401870, -2.555374, -0.755145, 1.570796, 1.630726],accel_mss,speed_ms,0,blend_radius_m)
    |   movel([0.060009, -1.401625, -2.555555, -0.755210, 1.570796, 1.630805],accel_mss,speed_ms,0,blend_radius_m)
    |   movel([0.060224, -1.401087, -2.555950, -0.755352, 1.570796, 1.631021],accel_mss,speed_ms,0,blend_radius_m)
    |   movel([0.060493, -1.400448, -2.556420, -0.755521, 1.570796, 1.631289],accel_mss,speed_ms,0,blend_radius_m)
    |   movel([0.060788, -1.399765, -2.556922, -0.755702, 1.570796, 1.631585],accel_mss,speed_ms,0,blend_radius_m)
    |   movel([0.061133, -1.398969, -2.557505, -0.755914, 1.570796, 1.631930],accel_mss,speed_ms,0,blend_radius_m)
    |   movel([0.061337, -1.398439, -2.557893, -0.756056, 1.570796, 1.632133],accel_mss,speed_ms,0,blend_radius_m)
    |   movel([0.061454, -1.398078, -2.558158, -0.756153, 1.570796, 1.632251],accel_mss,speed_ms,0,blend_radius_m)
    |   movel([0.061019, -1.398029, -2.558194, -0.756166, 1.570796, 1.631815],accel_mss,speed_ms,0,blend_radius_m)
    |   movel([0.060642, -1.398119, -2.558128, -0.756142, 1.570796, 1.631439],accel_mss,speed_ms,0,blend_radius_m)
    |   movel([0.060216, -1.398240, -2.558039, -0.756110, 1.570796, 1.631012],accel_mss,speed_ms,0,blend_radius_m)
    |   movel([0.059698, -1.398392, -2.557928, -0.756069, 1.570796, 1.630495],accel_mss,speed_ms,0,blend_radius_m)
    |   movel([0.059366, -1.398468, -2.557872, -0.756048, 1.570796, 1.630163],accel_mss,speed_ms,0,blend_radius_m)
    |   movel([0.059079, -1.398450, -2.557886, -0.756053, 1.570796, 1.629876],accel_mss,speed_ms,0,blend_radius_m)
    |   movel([0.059092, -1.398236, -2.558042, -0.756111, 1.570796, 1.629888],accel_mss,speed_ms,0,blend_radius_m)
    |   movel([0.060017, -1.396090, -2.559609, -0.756690, 1.570796, 1.630814],accel_mss,speed_ms,0,blend_radius_m)
    |   movel([0.060930, -1.394011, -2.561120, -0.757257, 1.570796, 1.631726],accel_mss,speed_ms,0,blend_radius_m)
    |   movel([0.061192, -1.393589, -2.561427, -0.757373, 1.570796, 1.631988],accel_mss,speed_ms,0,blend_radius_m)
    |   movel([0.061540, -1.393345, -2.561603, -0.757441, 1.570796, 1.632337],accel_mss,speed_ms,0,blend_radius_m)
    |   movel([0.062944, -1.392901, -2.561925, -0.757563, 1.570796, 1.633740],accel_mss,speed_ms,0,blend_radius_m)
    |   movel([0.064361, -1.392491, -2.562222, -0.757677, 1.570796, 1.635157],accel_mss,speed_ms,0,blend_radius_m)
    |   movel([0.064589, -1.392563, -2.562170, -0.757657, 1.570796, 1.635386],accel_mss,speed_ms,0,blend_radius_m)
    |   movel([0.064344, -1.393128, -2.561761, -0.757500, 1.570796, 1.635140],accel_mss,speed_ms,0,blend_radius_m)
    |   movel([0.064044, -1.393674, -2.561365, -0.757350, 1.570796, 1.634841],accel_mss,speed_ms,0,blend_radius_m)
    |   movel([0.063677, -1.394295, -2.560914, -0.757179, 1.570796, 1.634473],accel_mss,speed_ms,0,blend_radius_m)
    |   movel([0.063211, -1.395079, -2.560345, -0.756965, 1.570796, 1.634008],accel_mss,speed_ms,0,blend_radius_m)
    |   movel([0.062949, -1.395564, -2.559992, -0.756833, 1.570796, 1.633745],accel_mss,speed_ms,0,blend_radius_m)
    |   movel([0.062813, -1.395875, -2.559766, -0.756748, 1.570796, 1.633609],accel_mss,speed_ms,0,blend_radius_m)
    |   movel([0.062935, -1.396016, -2.559663, -0.756710, 1.570796, 1.633731],accel_mss,speed_ms,0,blend_radius_m)
    |   movel([0.063451, -1.395925, -2.559730, -0.756735, 1.570796, 1.634248],accel_mss,speed_ms,0,blend_radius_m)
    |   movel([0.063842, -1.395815, -2.559810, -0.756765, 1.570796, 1.634639],accel_mss,speed_ms,0,blend_radius_m)
    |   movel([0.064395, -1.395656, -2.559925, -0.756808, 1.570796, 1.635192],accel_mss,speed_ms,0,blend_radius_m)
    |   movel([0.064683, -1.395604, -2.559963, -0.756822, 1.570796, 1.635479],accel_mss,speed_ms,0,blend_radius_m)
    |   movel([0.064876, -1.395721, -2.559878, -0.756790, 1.570796, 1.635673],accel_mss,speed_ms,0,blend_radius_m)
    |   movel([0.064221, -1.396630, -2.559216, -0.756544, 1.570796, 1.635017],accel_mss,speed_ms,0,blend_radius_m)
    |   movel([0.063503, -1.397583, -2.558520, -0.756286, 1.570796, 1.634299],accel_mss,speed_ms,0,blend_radius_m)
    |   speed_ms = 0.003
    |   movel([0.063503, -1.400828, -2.559978, -0.751583, 1.570796, 1.634299],accel_mss,speed_ms,0,blend_radius_m)
    |   speed_ms = 0.007
    |   movel([0.062657, -1.401936, -2.559164, -0.751289, 1.570796, 1.633454],accel_mss,speed_ms,0,blend_radius_m)
    |   movel([0.061791, -1.403061, -2.558335, -0.750993, 1.570796, 1.632587],accel_mss,speed_ms,0,blend_radius_m)
    |   movel([0.061009, -1.404066, -2.557593, -0.750730, 1.570796, 1.631805],accel_mss,speed_ms,0,blend_radius_m)
    |   movel([0.060348, -1.404908, -2.556969, -0.750511, 1.570796, 1.631144],accel_mss,speed_ms,0,blend_radius_m)
    |   movel([0.060139, -1.405153, -2.556788, -0.750448, 1.570796, 1.630935],accel_mss,speed_ms,0,blend_radius_m)
    |   movel([0.059822, -1.405501, -2.556530, -0.750358, 1.570796, 1.630619],accel_mss,speed_ms,0,blend_radius_m)
    |   movel([0.059929, -1.405103, -2.556825, -0.750461, 1.570796, 1.630726],accel_mss,speed_ms,0,blend_radius_m)
    |   movel([0.060009, -1.404859, -2.557006, -0.750524, 1.570796, 1.630805],accel_mss,speed_ms,0,blend_radius_m)
    |   movel([0.060224, -1.404323, -2.557403, -0.750664, 1.570796, 1.631021],accel_mss,speed_ms,0,blend_radius_m)
    |   movel([0.060493, -1.403685, -2.557874, -0.750830, 1.570796, 1.631289],accel_mss,speed_ms,0,blend_radius_m)
    |   movel([0.060788, -1.403005, -2.558376, -0.751008, 1.570796, 1.631585],accel_mss,speed_ms,0,blend_radius_m)
    |   movel([0.061133, -1.402211, -2.558961, -0.751217, 1.570796, 1.631930],accel_mss,speed_ms,0,blend_radius_m)
    |   movel([0.061337, -1.401683, -2.559350, -0.751356, 1.570796, 1.632133],accel_mss,speed_ms,0,blend_radius_m)
    |   movel([0.061454, -1.401322, -2.559615, -0.751452, 1.570796, 1.632251],accel_mss,speed_ms,0,blend_radius_m)
    |   movel([0.061019, -1.401273, -2.559651, -0.751465, 1.570796, 1.631815],accel_mss,speed_ms,0,blend_radius_m)
    |   movel([0.060642, -1.401363, -2.559585, -0.751441, 1.570796, 1.631439],accel_mss,speed_ms,0,blend_radius_m)
    |   movel([0.060216, -1.401484, -2.559496, -0.751409, 1.570796, 1.631012],accel_mss,speed_ms,0,blend_radius_m)
    |   movel([0.059698, -1.401635, -2.559385, -0.751369, 1.570796, 1.630495],accel_mss,speed_ms,0,blend_radius_m)
    |   movel([0.059366, -1.401711, -2.559329, -0.751349, 1.570796, 1.630163],accel_mss,speed_ms,0,blend_radius_m)
    |   movel([0.059079, -1.401693, -2.559342, -0.751354, 1.570796, 1.629876],accel_mss,speed_ms,0,blend_radius_m)
    |   movel([0.059092, -1.401480, -2.559499, -0.751410, 1.570796, 1.629888],accel_mss,speed_ms,0,blend_radius_m)
    |   movel([0.060017, -1.399340, -2.561069, -0.751980, 1.570796, 1.630814],accel_mss,speed_ms,0,blend_radius_m)
    |   movel([0.060930, -1.397267, -2.562584, -0.752538, 1.570796, 1.631726],accel_mss,speed_ms,0,blend_radius_m)
    |   movel([0.061192, -1.396846, -2.562891, -0.752652, 1.570796, 1.631988],accel_mss,speed_ms,0,blend_radius_m)
    |   movel([0.061540, -1.396603, -2.563068, -0.752718, 1.570796, 1.632337],accel_mss,speed_ms,0,blend_radius_m)
    |   movel([0.062944, -1.396159, -2.563391, -0.752839, 1.570796, 1.633740],accel_mss,speed_ms,0,blend_radius_m)
    |   movel([0.064361, -1.395750, -2.563688, -0.752951, 1.570796, 1.635157],accel_mss,speed_ms,0,blend_radius_m)
    |   movel([0.064589, -1.395822, -2.563636, -0.752931, 1.570796, 1.635386],accel_mss,speed_ms,0,blend_radius_m)
    |   movel([0.064344, -1.396386, -2.563226, -0.752777, 1.570796, 1.635140],accel_mss,speed_ms,0,blend_radius_m)
    |   movel([0.064044, -1.396930, -2.562829, -0.752629, 1.570796, 1.634841],accel_mss,speed_ms,0,blend_radius_m)
    |   movel([0.063677, -1.397550, -2.562377, -0.752461, 1.570796, 1.634473],accel_mss,speed_ms,0,blend_radius_m)
    |   movel([0.063211, -1.398332, -2.561807, -0.752250, 1.570796, 1.634008],accel_mss,speed_ms,0,blend_radius_m)
    |   movel([0.062949, -1.398815, -2.561453, -0.752121, 1.570796, 1.633745],accel_mss,speed_ms,0,blend_radius_m)
    |   movel([0.062813, -1.399125, -2.561227, -0.752037, 1.570796, 1.633609],accel_mss,speed_ms,0,blend_radius_m)
    |   movel([0.062935, -1.399266, -2.561124, -0.752000, 1.570796, 1.633731],accel_mss,speed_ms,0,blend_radius_m)
    |   movel([0.063451, -1.399175, -2.561190, -0.752024, 1.570796, 1.634248],accel_mss,speed_ms,0,blend_radius_m)
    |   movel([0.063842, -1.399065, -2.561270, -0.752053, 1.570796, 1.634639],accel_mss,speed_ms,0,blend_radius_m)
    |   movel([0.064395, -1.398907, -2.561386, -0.752096, 1.570796, 1.635192],accel_mss,speed_ms,0,blend_radius_m)
    |   movel([0.064683, -1.398855, -2.561424, -0.752110, 1.570796, 1.635479],accel_mss,speed_ms,0,blend_radius_m)
    |   movel([0.064876, -1.398972, -2.561339, -0.752078, 1.570796, 1.635673],accel_mss,speed_ms,0,blend_radius_m)
    |   movel([0.064221, -1.399878, -2.560675, -0.751836, 1.570796, 1.635017],accel_mss,speed_ms,0,blend_radius_m)
    |   movel([0.063503, -1.400828, -2.559978, -0.751583, 1.570796, 1.634299],accel_mss,speed_ms,0,blend_radius_m)
    |   speed_ms = 0.003
    |   movel([0.063503, -1.387975, -2.554096, -0.770318, 1.570796, 1.634299],accel_mss,speed_ms,0,blend_radius_m)
    |   speed_ms = 1.000
    |   movel([0.063503, -1.363293, -2.541937, -0.807159, 1.570796, 1.634299],accel_mss,speed_ms,0,blend_radius_m)
    |   movel([0.062863, -1.377671, -2.531815, -0.802904, 1.570796, 1.633660],accel_mss,speed_ms,0,blend_radius_m)
    |   movel([0.062863, -1.402084, -2.543793, -0.766512, 1.570796, 1.633660],accel_mss,speed_ms,0,blend_radius_m)
    |   speed_ms = 0.003
    |   movel([0.062863, -1.411578, -2.548149, -0.752661, 1.570796, 1.633660],accel_mss,speed_ms,0,blend_radius_m)
    |   speed_ms = 0.007
    |   movel([0.063218, -1.411632, -2.548109, -0.752648, 1.570796, 1.634015],accel_mss,speed_ms,0,blend_radius_m)
    |   movel([0.063405, -1.411914, -2.547897, -0.752578, 1.570796, 1.634201],accel_mss,speed_ms,0,blend_radius_m)
    |   movel([0.063248, -1.412152, -2.547718, -0.752519, 1.570796, 1.634044],accel_mss,speed_ms,0,blend_radius_m)
    |   movel([0.062871, -1.412104, -2.547754, -0.752531, 1.570796, 1.633668],accel_mss,speed_ms,0,blend_radius_m)
    |   movel([0.062710, -1.411830, -2.547961, -0.752599, 1.570796, 1.633506],accel_mss,speed_ms,0,blend_radius_m)
    |   movel([0.062863, -1.411578, -2.548149, -0.752661, 1.570796, 1.633660],accel_mss,speed_ms,0,blend_radius_m)
    |   speed_ms = 0.003
    |   movel([0.062863, -1.414785, -2.549585, -0.748020, 1.570796, 1.633660],accel_mss,speed_ms,0,blend_radius_m)
    |   speed_ms = 0.007
    |   movel([0.063218, -1.414838, -2.549545, -0.748007, 1.570796, 1.634015],accel_mss,speed_ms,0,blend_radius_m)
    |   movel([0.063405, -1.415119, -2.549332, -0.747938, 1.570796, 1.634201],accel_mss,speed_ms,0,blend_radius_m)
    |   movel([0.063248, -1.415357, -2.549152, -0.747880, 1.570796, 1.634044],accel_mss,speed_ms,0,blend_radius_m)
    |   movel([0.062871, -1.415308, -2.549189, -0.747892, 1.570796, 1.633668],accel_mss,speed_ms,0,blend_radius_m)
    |   movel([0.062710, -1.415035, -2.549396, -0.747958, 1.570796, 1.633506],accel_mss,speed_ms,0,blend_radius_m)
    |   movel([0.062863, -1.414785, -2.549585, -0.748020, 1.570796, 1.633660],accel_mss,speed_ms,0,blend_radius_m)
    |   speed_ms = 0.003
    |   movel([0.062863, -1.402084, -2.543793, -0.766512, 1.570796, 1.633660],accel_mss,speed_ms,0,blend_radius_m)
    |   speed_ms = 1.000
    |   movel([0.062863, -1.377671, -2.531815, -0.802904, 1.570796, 1.633660],accel_mss,speed_ms,0,blend_radius_m)
    |   movel([0.065153, -1.377293, -2.532084, -0.803012, 1.570796, 1.635950],accel_mss,speed_ms,0,blend_radius_m)
    |   movel([0.065153, -1.401714, -2.544067, -0.766608, 1.570796, 1.635950],accel_mss,speed_ms,0,blend_radius_m)
    |   speed_ms = 0.003
    |   movel([0.065153, -1.411212, -2.548425, -0.752753, 1.570796, 1.635950],accel_mss,speed_ms,0,blend_radius_m)
    |   speed_ms = 0.007
    |   movel([0.065386, -1.410883, -2.548672, -0.752835, 1.570796, 1.636183],accel_mss,speed_ms,0,blend_radius_m)
    |   movel([0.065597, -1.411023, -2.548566, -0.752800, 1.570796, 1.636394],accel_mss,speed_ms,0,blend_radius_m)
    |   movel([0.065407, -1.411321, -2.548343, -0.752725, 1.570796, 1.636203],accel_mss,speed_ms,0,blend_radius_m)
    |   movel([0.065154, -1.411355, -2.548317, -0.752717, 1.570796, 1.635950],accel_mss,speed_ms,0,blend_radius_m)
    |   speed_ms = 0.003
    |   movel([0.065153, -1.414419, -2.549861, -0.748109, 1.570796, 1.635950],accel_mss,speed_ms,0,blend_radius_m)
    |   speed_ms = 0.007
    |   movel([0.065386, -1.414091, -2.550108, -0.748190, 1.570796, 1.636183],accel_mss,speed_ms,0,blend_radius_m)
    |   movel([0.065597, -1.414231, -2.550003, -0.748156, 1.570796, 1.636394],accel_mss,speed_ms,0,blend_radius_m)
    |   movel([0.065407, -1.414528, -2.549778, -0.748083, 1.570796, 1.636203],accel_mss,speed_ms,0,blend_radius_m)
    |   movel([0.065154, -1.414562, -2.549753, -0.748074, 1.570796, 1.635950],accel_mss,speed_ms,0,blend_radius_m)
    |   speed_ms = 0.003
    |   movel([0.065153, -1.401714, -2.544067, -0.766608, 1.570796, 1.635950],accel_mss,speed_ms,0,blend_radius_m)
    |   speed_ms = 1.000
    |   movel([0.065153, -1.377293, -2.532084, -0.803012, 1.570796, 1.635950],accel_mss,speed_ms,0,blend_radius_m)
    |   movel([0.064675, -1.377498, -2.531938, -0.802953, 1.570796, 1.635472],accel_mss,speed_ms,0,blend_radius_m)
    |   movel([0.064675, -1.401914, -2.543918, -0.766556, 1.570796, 1.635472],accel_mss,speed_ms,0,blend_radius_m)
    |   speed_ms = 0.003
    |   movel([0.064675, -1.411410, -2.548276, -0.752703, 1.570796, 1.635472],accel_mss,speed_ms,0,blend_radius_m)
    |   speed_ms = 0.007
    |   movel([0.064499, -1.411772, -2.548004, -0.752613, 1.570796, 1.635295],accel_mss,speed_ms,0,blend_radius_m)
    |   movel([0.064240, -1.411944, -2.547875, -0.752570, 1.570796, 1.635037],accel_mss,speed_ms,0,blend_radius_m)
    |   movel([0.063993, -1.411883, -2.547920, -0.752586, 1.570796, 1.634789],accel_mss,speed_ms,0,blend_radius_m)
    |   movel([0.063850, -1.411583, -2.548146, -0.752660, 1.570796, 1.634646],accel_mss,speed_ms,0,blend_radius_m)
    |   movel([0.063694, -1.411303, -2.548356, -0.752730, 1.570796, 1.634490],accel_mss,speed_ms,0,blend_radius_m)
    |   movel([0.063381, -1.411164, -2.548461, -0.752765, 1.570796, 1.634177],accel_mss,speed_ms,0,blend_radius_m)
    |   movel([0.062972, -1.411194, -2.548438, -0.752757, 1.570796, 1.633768],accel_mss,speed_ms,0,blend_radius_m)
    |   movel([0.062556, -1.411383, -2.548296, -0.752710, 1.570796, 1.633353],accel_mss,speed_ms,0,blend_radius_m)
    |   movel([0.062327, -1.411575, -2.548152, -0.752662, 1.570796, 1.633124],accel_mss,speed_ms,0,blend_radius_m)
    |   movel([0.062153, -1.411988, -2.547841, -0.752559, 1.570796, 1.632949],accel_mss,speed_ms,0,blend_radius_m)
    |   movel([0.062221, -1.412182, -2.547696, -0.752511, 1.570796, 1.633018],accel_mss,speed_ms,0,blend_radius_m)
    |   movel([0.062392, -1.412391, -2.547538, -0.752460, 1.570796, 1.633189],accel_mss,speed_ms,0,blend_radius_m)
    |   movel([0.062579, -1.412520, -2.547441, -0.752428, 1.570796, 1.633375],accel_mss,speed_ms,0,blend_radius_m)
    |   movel([0.062801, -1.412574, -2.547401, -0.752414, 1.570796, 1.633597],accel_mss,speed_ms,0,blend_radius_m)
    |   movel([0.063075, -1.412565, -2.547408, -0.752417, 1.570796, 1.633872],accel_mss,speed_ms,0,blend_radius_m)
    |   movel([0.063305, -1.412551, -2.547418, -0.752420, 1.570796, 1.634102],accel_mss,speed_ms,0,blend_radius_m)
    |   movel([0.063464, -1.412724, -2.547288, -0.752377, 1.570796, 1.634261],accel_mss,speed_ms,0,blend_radius_m)
    |   movel([0.063488, -1.413068, -2.547029, -0.752292, 1.570796, 1.634284],accel_mss,speed_ms,0,blend_radius_m)
    |   movel([0.063495, -1.413351, -2.546815, -0.752223, 1.570796, 1.634291],accel_mss,speed_ms,0,blend_radius_m)
    |   movel([0.063493, -1.413759, -2.546508, -0.752123, 1.570796, 1.634289],accel_mss,speed_ms,0,blend_radius_m)
    |   movel([0.063485, -1.414205, -2.546171, -0.752013, 1.570796, 1.634281],accel_mss,speed_ms,0,blend_radius_m)
    |   movel([0.063470, -1.414632, -2.545848, -0.751909, 1.570796, 1.634266],accel_mss,speed_ms,0,blend_radius_m)
    |   movel([0.063440, -1.415216, -2.545407, -0.751766, 1.570796, 1.634236],accel_mss,speed_ms,0,blend_radius_m)
    |   movel([0.063398, -1.415485, -2.545203, -0.751701, 1.570796, 1.634195],accel_mss,speed_ms,0,blend_radius_m)
    |   movel([0.063213, -1.415734, -2.545014, -0.751641, 1.570796, 1.634009],accel_mss,speed_ms,0,blend_radius_m)
    |   movel([0.062987, -1.415735, -2.545014, -0.751640, 1.570796, 1.633784],accel_mss,speed_ms,0,blend_radius_m)
    |   movel([0.062901, -1.415541, -2.545160, -0.751687, 1.570796, 1.633697],accel_mss,speed_ms,0,blend_radius_m)
    |   movel([0.062816, -1.415322, -2.545327, -0.751741, 1.570796, 1.633612],accel_mss,speed_ms,0,blend_radius_m)
    |   movel([0.062809, -1.415093, -2.545500, -0.751796, 1.570796, 1.633606],accel_mss,speed_ms,0,blend_radius_m)
    |   movel([0.062628, -1.414808, -2.545715, -0.751866, 1.570796, 1.633425],accel_mss,speed_ms,0,blend_radius_m)
    |   movel([0.062390, -1.414746, -2.545762, -0.751881, 1.570796, 1.633187],accel_mss,speed_ms,0,blend_radius_m)
    |   movel([0.062139, -1.414777, -2.545739, -0.751873, 1.570796, 1.632935],accel_mss,speed_ms,0,blend_radius_m)
    |   movel([0.061709, -1.414792, -2.545727, -0.751870, 1.570796, 1.632506],accel_mss,speed_ms,0,blend_radius_m)
    |   movel([0.061418, -1.414755, -2.545756, -0.751879, 1.570796, 1.632214],accel_mss,speed_ms,0,blend_radius_m)
    |   movel([0.061133, -1.414693, -2.545802, -0.751894, 1.570796, 1.631929],accel_mss,speed_ms,0,blend_radius_m)
    |   movel([0.060182, -1.414220, -2.546159, -0.752009, 1.570796, 1.630978],accel_mss,speed_ms,0,blend_radius_m)
    |   movel([0.059674, -1.413438, -2.546749, -0.752201, 1.570796, 1.630470],accel_mss,speed_ms,0,blend_radius_m)
    |   movel([0.059654, -1.412389, -2.547540, -0.752460, 1.570796, 1.630450],accel_mss,speed_ms,0,blend_radius_m)
    |   movel([0.060113, -1.411143, -2.548476, -0.752770, 1.570796, 1.630909],accel_mss,speed_ms,0,blend_radius_m)
    |   movel([0.060729, -1.410205, -2.549180, -0.753004, 1.570796, 1.631525],accel_mss,speed_ms,0,blend_radius_m)
    |   movel([0.061542, -1.409345, -2.549823, -0.753220, 1.570796, 1.632338],accel_mss,speed_ms,0,blend_radius_m)
    |   movel([0.062503, -1.408612, -2.550372, -0.753405, 1.570796, 1.633300],accel_mss,speed_ms,0,blend_radius_m)
    |   movel([0.063563, -1.408046, -2.550794, -0.753549, 1.570796, 1.634359],accel_mss,speed_ms,0,blend_radius_m)
    |   movel([0.065284, -1.407542, -2.551170, -0.753677, 1.570796, 1.636081],accel_mss,speed_ms,0,blend_radius_m)
    |   movel([0.066894, -1.407547, -2.551166, -0.753676, 1.570796, 1.637690],accel_mss,speed_ms,0,blend_radius_m)
    |   movel([0.068166, -1.408046, -2.550794, -0.753549, 1.570796, 1.638962],accel_mss,speed_ms,0,blend_radius_m)
    |   movel([0.068919, -1.408979, -2.550098, -0.753313, 1.570796, 1.639715],accel_mss,speed_ms,0,blend_radius_m)
    |   movel([0.069004, -1.409463, -2.549735, -0.753191, 1.570796, 1.639801],accel_mss,speed_ms,0,blend_radius_m)
    |   movel([0.068940, -1.410222, -2.549167, -0.753000, 1.570796, 1.639737],accel_mss,speed_ms,0,blend_radius_m)
    |   movel([0.068780, -1.410999, -2.548584, -0.752805, 1.570796, 1.639577],accel_mss,speed_ms,0,blend_radius_m)
    |   movel([0.068544, -1.411554, -2.548167, -0.752667, 1.570796, 1.639341],accel_mss,speed_ms,0,blend_radius_m)
    |   movel([0.068055, -1.412218, -2.547668, -0.752502, 1.570796, 1.638851],accel_mss,speed_ms,0,blend_radius_m)
    |   movel([0.067404, -1.412843, -2.547198, -0.752348, 1.570796, 1.638201],accel_mss,speed_ms,0,blend_radius_m)
    |   movel([0.066687, -1.413344, -2.546821, -0.752225, 1.570796, 1.637483],accel_mss,speed_ms,0,blend_radius_m)
    |   movel([0.066009, -1.413641, -2.546596, -0.752151, 1.570796, 1.636805],accel_mss,speed_ms,0,blend_radius_m)
    |   movel([0.065633, -1.413791, -2.546483, -0.752115, 1.570796, 1.636429],accel_mss,speed_ms,0,blend_radius_m)
    |   movel([0.065392, -1.413955, -2.546359, -0.752074, 1.570796, 1.636188],accel_mss,speed_ms,0,blend_radius_m)
    |   movel([0.065244, -1.414196, -2.546178, -0.752015, 1.570796, 1.636040],accel_mss,speed_ms,0,blend_radius_m)
    |   movel([0.065148, -1.414497, -2.545950, -0.751942, 1.570796, 1.635944],accel_mss,speed_ms,0,blend_radius_m)
    |   movel([0.065119, -1.414780, -2.545736, -0.751873, 1.570796, 1.635915],accel_mss,speed_ms,0,blend_radius_m)
    |   movel([0.065175, -1.414969, -2.545594, -0.751827, 1.570796, 1.635971],accel_mss,speed_ms,0,blend_radius_m)
    |   movel([0.065137, -1.415185, -2.545430, -0.751774, 1.570796, 1.635933],accel_mss,speed_ms,0,blend_radius_m)
    |   movel([0.064504, -1.415374, -2.545287, -0.751728, 1.570796, 1.635301],accel_mss,speed_ms,0,blend_radius_m)
    |   movel([0.064550, -1.414566, -2.545898, -0.751925, 1.570796, 1.635346],accel_mss,speed_ms,0,blend_radius_m)
    |   movel([0.064576, -1.414252, -2.546135, -0.752002, 1.570796, 1.635372],accel_mss,speed_ms,0,blend_radius_m)
    |   movel([0.064615, -1.413983, -2.546338, -0.752067, 1.570796, 1.635412],accel_mss,speed_ms,0,blend_radius_m)
    |   movel([0.064662, -1.413768, -2.546501, -0.752120, 1.570796, 1.635459],accel_mss,speed_ms,0,blend_radius_m)
    |   movel([0.064796, -1.413502, -2.546702, -0.752186, 1.570796, 1.635592],accel_mss,speed_ms,0,blend_radius_m)
    |   movel([0.064830, -1.413276, -2.546871, -0.752241, 1.570796, 1.635626],accel_mss,speed_ms,0,blend_radius_m)
    |   movel([0.064847, -1.413014, -2.547069, -0.752306, 1.570796, 1.635644],accel_mss,speed_ms,0,blend_radius_m)
    |   movel([0.064875, -1.412339, -2.547578, -0.752473, 1.570796, 1.635672],accel_mss,speed_ms,0,blend_radius_m)
    |   movel([0.065408, -1.411823, -2.547966, -0.752601, 1.570796, 1.636204],accel_mss,speed_ms,0,blend_radius_m)
    |   movel([0.065763, -1.411443, -2.548251, -0.752695, 1.570796, 1.636560],accel_mss,speed_ms,0,blend_radius_m)
    |   movel([0.065967, -1.411133, -2.548484, -0.752772, 1.570796, 1.636763],accel_mss,speed_ms,0,blend_radius_m)
    |   movel([0.066037, -1.410862, -2.548687, -0.752840, 1.570796, 1.636834],accel_mss,speed_ms,0,blend_radius_m)
    |   movel([0.065994, -1.410600, -2.548883, -0.752905, 1.570796, 1.636790],accel_mss,speed_ms,0,blend_radius_m)
    |   movel([0.065732, -1.410421, -2.549018, -0.752950, 1.570796, 1.636528],accel_mss,speed_ms,0,blend_radius_m)
    |   movel([0.065334, -1.410524, -2.548941, -0.752924, 1.570796, 1.636130],accel_mss,speed_ms,0,blend_radius_m)
    |   movel([0.064927, -1.410902, -2.548657, -0.752830, 1.570796, 1.635723],accel_mss,speed_ms,0,blend_radius_m)
    |   movel([0.064675, -1.411410, -2.548276, -0.752703, 1.570796, 1.635472],accel_mss,speed_ms,0,blend_radius_m)
    |   speed_ms = 0.003
    |   movel([0.064675, -1.414617, -2.549711, -0.748061, 1.570796, 1.635472],accel_mss,speed_ms,0,blend_radius_m)
    |   speed_ms = 0.007
    |   movel([0.064499, -1.414977, -2.549439, -0.747972, 1.570796, 1.635295],accel_mss,speed_ms,0,blend_radius_m)
    |   movel([0.064240, -1.415149, -2.549309, -0.747931, 1.570796, 1.635037],accel_mss,speed_ms,0,blend_radius_m)
    |   movel([0.063993, -1.415088, -2.549355, -0.747945, 1.570796, 1.634789],accel_mss,speed_ms,0,blend_radius_m)
    |   movel([0.063850, -1.414789, -2.549581, -0.748019, 1.570796, 1.634646],accel_mss,speed_ms,0,blend_radius_m)
    |   movel([0.063694, -1.414510, -2.549792, -0.748087, 1.570796, 1.634490],accel_mss,speed_ms,0,blend_radius_m)
    |   movel([0.063381, -1.414371, -2.549897, -0.748121, 1.570796, 1.634177],accel_mss,speed_ms,0,blend_radius_m)
    |   movel([0.062972, -1.414402, -2.549874, -0.748114, 1.570796, 1.633768],accel_mss,speed_ms,0,blend_radius_m)
    |   movel([0.062556, -1.414590, -2.549732, -0.748067, 1.570796, 1.633353],accel_mss,speed_ms,0,blend_radius_m)
    |   movel([0.062327, -1.414781, -2.549587, -0.748020, 1.570796, 1.633124],accel_mss,speed_ms,0,blend_radius_m)
    |   movel([0.062153, -1.415193, -2.549276, -0.747920, 1.570796, 1.632949],accel_mss,speed_ms,0,blend_radius_m)
    |   movel([0.062221, -1.415386, -2.549130, -0.747873, 1.570796, 1.633018],accel_mss,speed_ms,0,blend_radius_m)
    |   movel([0.062392, -1.415595, -2.548972, -0.747822, 1.570796, 1.633189],accel_mss,speed_ms,0,blend_radius_m)
    |   movel([0.062579, -1.415723, -2.548875, -0.747790, 1.570796, 1.633375],accel_mss,speed_ms,0,blend_radius_m)
    |   movel([0.062801, -1.415777, -2.548835, -0.747777, 1.570796, 1.633597],accel_mss,speed_ms,0,blend_radius_m)
    |   movel([0.063075, -1.415768, -2.548841, -0.747779, 1.570796, 1.633872],accel_mss,speed_ms,0,blend_radius_m)
    |   movel([0.063305, -1.415754, -2.548852, -0.747783, 1.570796, 1.634102],accel_mss,speed_ms,0,blend_radius_m)
    |   movel([0.063464, -1.415927, -2.548722, -0.747741, 1.570796, 1.634261],accel_mss,speed_ms,0,blend_radius_m)
    |   movel([0.063488, -1.416270, -2.548462, -0.747658, 1.570796, 1.634284],accel_mss,speed_ms,0,blend_radius_m)
    |   movel([0.063495, -1.416552, -2.548248, -0.747589, 1.570796, 1.634291],accel_mss,speed_ms,0,blend_radius_m)
    |   movel([0.063493, -1.416959, -2.547940, -0.747491, 1.570796, 1.634289],accel_mss,speed_ms,0,blend_radius_m)
    |   movel([0.063485, -1.417404, -2.547602, -0.747383, 1.570796, 1.634281],accel_mss,speed_ms,0,blend_radius_m)
    |   movel([0.063470, -1.417829, -2.547279, -0.747281, 1.570796, 1.634266],accel_mss,speed_ms,0,blend_radius_m)
    |   movel([0.063440, -1.418412, -2.546836, -0.747141, 1.570796, 1.634236],accel_mss,speed_ms,0,blend_radius_m)
    |   movel([0.063398, -1.418680, -2.546632, -0.747077, 1.570796, 1.634195],accel_mss,speed_ms,0,blend_radius_m)
    |   movel([0.063213, -1.418928, -2.546443, -0.747018, 1.570796, 1.634009],accel_mss,speed_ms,0,blend_radius_m)
    |   movel([0.062987, -1.418929, -2.546443, -0.747017, 1.570796, 1.633784],accel_mss,speed_ms,0,blend_radius_m)
    |   movel([0.062901, -1.418736, -2.546589, -0.747063, 1.570796, 1.633697],accel_mss,speed_ms,0,blend_radius_m)
    |   movel([0.062816, -1.418517, -2.546756, -0.747116, 1.570796, 1.633612],accel_mss,speed_ms,0,blend_radius_m)
    |   movel([0.062809, -1.418289, -2.546930, -0.747171, 1.570796, 1.633606],accel_mss,speed_ms,0,blend_radius_m)
    |   movel([0.062628, -1.418005, -2.547146, -0.747239, 1.570796, 1.633425],accel_mss,speed_ms,0,blend_radius_m)
    |   movel([0.062390, -1.417943, -2.547192, -0.747253, 1.570796, 1.633187],accel_mss,speed_ms,0,blend_radius_m)
    |   movel([0.062139, -1.417974, -2.547169, -0.747246, 1.570796, 1.632935],accel_mss,speed_ms,0,blend_radius_m)
    |   movel([0.061709, -1.417989, -2.547158, -0.747242, 1.570796, 1.632506],accel_mss,speed_ms,0,blend_radius_m)
    |   movel([0.061418, -1.417952, -2.547186, -0.747251, 1.570796, 1.632214],accel_mss,speed_ms,0,blend_radius_m)
    |   movel([0.061133, -1.417891, -2.547232, -0.747266, 1.570796, 1.631929],accel_mss,speed_ms,0,blend_radius_m)
    |   movel([0.060182, -1.417419, -2.547590, -0.747380, 1.570796, 1.630978],accel_mss,speed_ms,0,blend_radius_m)
    |   movel([0.059674, -1.416639, -2.548182, -0.747568, 1.570796, 1.630470],accel_mss,speed_ms,0,blend_radius_m)
    |   movel([0.059654, -1.415593, -2.548974, -0.747822, 1.570796, 1.630450],accel_mss,speed_ms,0,blend_radius_m)
    |   movel([0.060113, -1.414350, -2.549912, -0.748126, 1.570796, 1.630909],accel_mss,speed_ms,0,blend_radius_m)
    |   movel([0.060729, -1.413415, -2.550618, -0.748357, 1.570796, 1.631525],accel_mss,speed_ms,0,blend_radius_m)
    |   movel([0.061542, -1.412558, -2.551262, -0.748569, 1.570796, 1.632338],accel_mss,speed_ms,0,blend_radius_m)
    |   movel([0.062503, -1.411826, -2.551812, -0.748751, 1.570796, 1.633300],accel_mss,speed_ms,0,blend_radius_m)
    |   movel([0.063563, -1.411262, -2.552235, -0.748892, 1.570796, 1.634359],accel_mss,speed_ms,0,blend_radius_m)
    |   movel([0.065284, -1.410760, -2.552611, -0.749017, 1.570796, 1.636081],accel_mss,speed_ms,0,blend_radius_m)
    |   movel([0.066894, -1.410764, -2.552608, -0.749016, 1.570796, 1.637690],accel_mss,speed_ms,0,blend_radius_m)
    |   movel([0.068166, -1.411262, -2.552235, -0.748892, 1.570796, 1.638962],accel_mss,speed_ms,0,blend_radius_m)
    |   movel([0.068919, -1.412192, -2.551537, -0.748660, 1.570796, 1.639715],accel_mss,speed_ms,0,blend_radius_m)
    |   movel([0.069004, -1.412675, -2.551174, -0.748540, 1.570796, 1.639801],accel_mss,speed_ms,0,blend_radius_m)
    |   movel([0.068940, -1.413432, -2.550605, -0.748352, 1.570796, 1.639737],accel_mss,speed_ms,0,blend_radius_m)
    |   movel([0.068780, -1.414207, -2.550020, -0.748161, 1.570796, 1.639577],accel_mss,speed_ms,0,blend_radius_m)
    |   movel([0.068544, -1.414760, -2.549603, -0.748026, 1.570796, 1.639341],accel_mss,speed_ms,0,blend_radius_m)
    |   movel([0.068055, -1.415423, -2.549103, -0.747864, 1.570796, 1.638851],accel_mss,speed_ms,0,blend_radius_m)
    |   movel([0.067404, -1.416046, -2.548631, -0.747712, 1.570796, 1.638201],accel_mss,speed_ms,0,blend_radius_m)
    |   movel([0.066687, -1.416545, -2.548253, -0.747591, 1.570796, 1.637483],accel_mss,speed_ms,0,blend_radius_m)
    |   movel([0.066009, -1.416842, -2.548028, -0.747519, 1.570796, 1.636805],accel_mss,speed_ms,0,blend_radius_m)
    |   movel([0.065633, -1.416991, -2.547915, -0.747483, 1.570796, 1.636429],accel_mss,speed_ms,0,blend_radius_m)
    |   movel([0.065392, -1.417155, -2.547791, -0.747443, 1.570796, 1.636188],accel_mss,speed_ms,0,blend_radius_m)
    |   movel([0.065244, -1.417395, -2.547609, -0.747385, 1.570796, 1.636040],accel_mss,speed_ms,0,blend_radius_m)
    |   movel([0.065148, -1.417695, -2.547381, -0.747313, 1.570796, 1.635944],accel_mss,speed_ms,0,blend_radius_m)
    |   movel([0.065119, -1.417977, -2.547167, -0.747245, 1.570796, 1.635915],accel_mss,speed_ms,0,blend_radius_m)
    |   movel([0.065175, -1.418165, -2.547024, -0.747200, 1.570796, 1.635971],accel_mss,speed_ms,0,blend_radius_m)
    |   movel([0.065137, -1.418381, -2.546860, -0.747149, 1.570796, 1.635933],accel_mss,speed_ms,0,blend_radius_m)
    |   movel([0.064504, -1.418569, -2.546717, -0.747103, 1.570796, 1.635301],accel_mss,speed_ms,0,blend_radius_m)
    |   movel([0.064550, -1.417764, -2.547329, -0.747297, 1.570796, 1.635346],accel_mss,speed_ms,0,blend_radius_m)
    |   movel([0.064576, -1.417450, -2.547567, -0.747372, 1.570796, 1.635372],accel_mss,speed_ms,0,blend_radius_m)
    |   movel([0.064615, -1.417183, -2.547770, -0.747437, 1.570796, 1.635412],accel_mss,speed_ms,0,blend_radius_m)
    |   movel([0.064662, -1.416968, -2.547933, -0.747488, 1.570796, 1.635459],accel_mss,speed_ms,0,blend_radius_m)
    |   movel([0.064796, -1.416702, -2.548134, -0.747553, 1.570796, 1.635592],accel_mss,speed_ms,0,blend_radius_m)
    |   movel([0.064830, -1.416478, -2.548304, -0.747607, 1.570796, 1.635626],accel_mss,speed_ms,0,blend_radius_m)
    |   movel([0.064847, -1.416216, -2.548503, -0.747671, 1.570796, 1.635644],accel_mss,speed_ms,0,blend_radius_m)
    |   movel([0.064875, -1.415543, -2.549012, -0.747834, 1.570796, 1.635672],accel_mss,speed_ms,0,blend_radius_m)
    |   movel([0.065408, -1.415028, -2.549401, -0.747960, 1.570796, 1.636204],accel_mss,speed_ms,0,blend_radius_m)
    |   movel([0.065763, -1.414649, -2.549687, -0.748053, 1.570796, 1.636560],accel_mss,speed_ms,0,blend_radius_m)
    |   movel([0.065967, -1.414340, -2.549920, -0.748129, 1.570796, 1.636763],accel_mss,speed_ms,0,blend_radius_m)
    |   movel([0.066037, -1.414070, -2.550124, -0.748195, 1.570796, 1.636834],accel_mss,speed_ms,0,blend_radius_m)
    |   movel([0.065994, -1.413809, -2.550320, -0.748259, 1.570796, 1.636790],accel_mss,speed_ms,0,blend_radius_m)
    |   movel([0.065732, -1.413630, -2.550455, -0.748303, 1.570796, 1.636528],accel_mss,speed_ms,0,blend_radius_m)
    |   movel([0.065334, -1.413733, -2.550378, -0.748278, 1.570796, 1.636130],accel_mss,speed_ms,0,blend_radius_m)
    |   movel([0.064927, -1.414110, -2.550094, -0.748185, 1.570796, 1.635723],accel_mss,speed_ms,0,blend_radius_m)
    |   movel([0.064675, -1.414617, -2.549711, -0.748061, 1.570796, 1.635472],accel_mss,speed_ms,0,blend_radius_m)
    |   speed_ms = 0.003
    |   movel([0.064675, -1.401914, -2.543918, -0.766556, 1.570796, 1.635472],accel_mss,speed_ms,0,blend_radius_m)
    |   speed_ms = 1.000
    |   movel([0.064675, -1.377498, -2.531938, -0.802953, 1.570796, 1.635472],accel_mss,speed_ms,0,blend_radius_m)
    |   movel([0.064357, -1.378354, -2.531327, -0.802708, 1.570796, 1.635153],accel_mss,speed_ms,0,blend_radius_m)
    |   movel([0.064357, -1.402754, -2.543296, -0.766339, 1.570796, 1.635153],accel_mss,speed_ms,0,blend_radius_m)
    |   speed_ms = 0.003
    |   movel([0.064357, -1.412243, -2.547649, -0.752496, 1.570796, 1.635153],accel_mss,speed_ms,0,blend_radius_m)
    |   speed_ms = 0.007
    |   movel([0.064463, -1.412398, -2.547533, -0.752458, 1.570796, 1.635259],accel_mss,speed_ms,0,blend_radius_m)
    |   movel([0.064395, -1.412789, -2.547239, -0.752361, 1.570796, 1.635192],accel_mss,speed_ms,0,blend_radius_m)
    |   movel([0.064340, -1.413059, -2.547035, -0.752295, 1.570796, 1.635136],accel_mss,speed_ms,0,blend_radius_m)
    |   movel([0.064277, -1.413476, -2.546721, -0.752192, 1.570796, 1.635074],accel_mss,speed_ms,0,blend_radius_m)
    |   movel([0.064218, -1.413944, -2.546368, -0.752077, 1.570796, 1.635014],accel_mss,speed_ms,0,blend_radius_m)
    |   movel([0.064174, -1.414403, -2.546021, -0.751965, 1.570796, 1.634970],accel_mss,speed_ms,0,blend_radius_m)
    |   movel([0.064132, -1.414826, -2.545702, -0.751861, 1.570796, 1.634929],accel_mss,speed_ms,0,blend_radius_m)
    |   movel([0.064077, -1.415186, -2.545429, -0.751774, 1.570796, 1.634873],accel_mss,speed_ms,0,blend_radius_m)
    |   movel([0.064019, -1.415486, -2.545202, -0.751701, 1.570796, 1.634815],accel_mss,speed_ms,0,blend_radius_m)
    |   movel([0.063912, -1.415161, -2.545448, -0.751780, 1.570796, 1.634708],accel_mss,speed_ms,0,blend_radius_m)
    |   movel([0.063906, -1.414739, -2.545767, -0.751883, 1.570796, 1.634702],accel_mss,speed_ms,0,blend_radius_m)
    |   movel([0.063919, -1.414229, -2.546152, -0.752007, 1.570796, 1.634715],accel_mss,speed_ms,0,blend_radius_m)
    |   movel([0.063935, -1.413704, -2.546549, -0.752136, 1.570796, 1.634731],accel_mss,speed_ms,0,blend_radius_m)
    |   movel([0.063935, -1.413240, -2.546899, -0.752250, 1.570796, 1.634731],accel_mss,speed_ms,0,blend_radius_m)
    |   movel([0.063924, -1.412854, -2.547190, -0.752345, 1.570796, 1.634720],accel_mss,speed_ms,0,blend_radius_m)
    |   movel([0.063863, -1.412666, -2.547331, -0.752392, 1.570796, 1.634659],accel_mss,speed_ms,0,blend_radius_m)
    |   movel([0.064138, -1.412460, -2.547487, -0.752443, 1.570796, 1.634934],accel_mss,speed_ms,0,blend_radius_m)
    |   movel([0.064357, -1.412243, -2.547649, -0.752496, 1.570796, 1.635153],accel_mss,speed_ms,0,blend_radius_m)
    |   speed_ms = 0.003
    |   movel([0.064357, -1.415448, -2.549084, -0.747858, 1.570796, 1.635153],accel_mss,speed_ms,0,blend_radius_m)
    |   speed_ms = 0.007
    |   movel([0.064463, -1.415602, -2.548967, -0.747820, 1.570796, 1.635259],accel_mss,speed_ms,0,blend_radius_m)
    |   movel([0.064395, -1.415992, -2.548672, -0.747725, 1.570796, 1.635192],accel_mss,speed_ms,0,blend_radius_m)
    |   movel([0.064340, -1.416261, -2.548468, -0.747660, 1.570796, 1.635136],accel_mss,speed_ms,0,blend_radius_m)
    |   movel([0.064277, -1.416677, -2.548153, -0.747559, 1.570796, 1.635074],accel_mss,speed_ms,0,blend_radius_m)
    |   movel([0.064218, -1.417144, -2.547799, -0.747446, 1.570796, 1.635014],accel_mss,speed_ms,0,blend_radius_m)
    |   movel([0.064174, -1.417602, -2.547452, -0.747336, 1.570796, 1.634970],accel_mss,speed_ms,0,blend_radius_m)
    |   movel([0.064132, -1.418023, -2.547132, -0.747234, 1.570796, 1.634929],accel_mss,speed_ms,0,blend_radius_m)
    |   movel([0.064077, -1.418382, -2.546859, -0.747148, 1.570796, 1.634873],accel_mss,speed_ms,0,blend_radius_m)
    |   movel([0.064019, -1.418681, -2.546631, -0.747077, 1.570796, 1.634815],accel_mss,speed_ms,0,blend_radius_m)
    |   movel([0.063912, -1.418357, -2.546878, -0.747154, 1.570796, 1.634708],accel_mss,speed_ms,0,blend_radius_m)
    |   movel([0.063906, -1.417936, -2.547198, -0.747255, 1.570796, 1.634702],accel_mss,speed_ms,0,blend_radius_m)
    |   movel([0.063919, -1.417428, -2.547584, -0.747377, 1.570796, 1.634715],accel_mss,speed_ms,0,blend_radius_m)
    |   movel([0.063935, -1.416905, -2.547981, -0.747504, 1.570796, 1.634731],accel_mss,speed_ms,0,blend_radius_m)
    |   movel([0.063935, -1.416441, -2.548332, -0.747616, 1.570796, 1.634731],accel_mss,speed_ms,0,blend_radius_m)
    |   movel([0.063924, -1.416056, -2.548623, -0.747709, 1.570796, 1.634720],accel_mss,speed_ms,0,blend_radius_m)
    |   movel([0.063863, -1.415869, -2.548765, -0.747755, 1.570796, 1.634659],accel_mss,speed_ms,0,blend_radius_m)
    |   movel([0.064138, -1.415663, -2.548921, -0.747805, 1.570796, 1.634934],accel_mss,speed_ms,0,blend_radius_m)
    |   movel([0.064357, -1.415448, -2.549084, -0.747858, 1.570796, 1.635153],accel_mss,speed_ms,0,blend_radius_m)
    |   speed_ms = 0.003
    |   movel([0.064357, -1.402754, -2.543296, -0.766339, 1.570796, 1.635153],accel_mss,speed_ms,0,blend_radius_m)
    |   speed_ms = 1.000
    |   movel([0.064357, -1.378354, -2.531327, -0.802708, 1.570796, 1.635153],accel_mss,speed_ms,0,blend_radius_m)
    |   movel([0.062676, -1.381664, -2.528953, -0.801772, 1.570796, 1.633472],accel_mss,speed_ms,0,blend_radius_m)
    |   movel([0.062676, -1.406002, -2.540881, -0.765506, 1.570796, 1.633472],accel_mss,speed_ms,0,blend_radius_m)
    |   speed_ms = 0.003
    |   movel([0.062676, -1.415464, -2.545219, -0.751706, 1.570796, 1.633472],accel_mss,speed_ms,0,blend_radius_m)
    |   speed_ms = 0.007
    |   speed_ms = 0.003
    |   movel([0.062676, -1.418659, -2.546648, -0.747082, 1.570796, 1.633472],accel_mss,speed_ms,0,blend_radius_m)
    |   speed_ms = 0.007
    |   speed_ms = 0.003
    |   movel([0.062676, -1.406002, -2.540881, -0.765506, 1.570796, 1.633472],accel_mss,speed_ms,0,blend_radius_m)
    |   speed_ms = 1.000
    |   movel([0.062676, -1.381664, -2.528953, -0.801772, 1.570796, 1.633472],accel_mss,speed_ms,0,blend_radius_m)
    |   movel([0.062527, -1.382550, -2.528315, -0.801524, 1.570796, 1.633324],accel_mss,speed_ms,0,blend_radius_m)
    |   movel([0.062527, -1.406871, -2.540231, -0.765286, 1.570796, 1.633324],accel_mss,speed_ms,0,blend_radius_m)
    |   speed_ms = 0.003
    |   movel([0.062527, -1.416327, -2.544565, -0.751497, 1.570796, 1.633324],accel_mss,speed_ms,0,blend_radius_m)
    |   speed_ms = 0.007
    |   movel([0.063795, -1.416027, -2.544793, -0.751570, 1.570796, 1.634591],accel_mss,speed_ms,0,blend_radius_m)
    |   movel([0.064285, -1.415913, -2.544879, -0.751597, 1.570796, 1.635081],accel_mss,speed_ms,0,blend_radius_m)
    |   movel([0.064715, -1.415821, -2.544948, -0.751619, 1.570796, 1.635511],accel_mss,speed_ms,0,blend_radius_m)
    |   movel([0.065077, -1.415747, -2.545004, -0.751637, 1.570796, 1.635874],accel_mss,speed_ms,0,blend_radius_m)
    |   movel([0.065199, -1.415936, -2.544861, -0.751592, 1.570796, 1.635995],accel_mss,speed_ms,0,blend_radius_m)
    |   movel([0.065192, -1.416358, -2.544542, -0.751490, 1.570796, 1.635988],accel_mss,speed_ms,0,blend_radius_m)
    |   movel([0.065156, -1.416670, -2.544305, -0.751414, 1.570796, 1.635953],accel_mss,speed_ms,0,blend_radius_m)
    |   movel([0.065014, -1.417051, -2.544016, -0.751323, 1.570796, 1.635811],accel_mss,speed_ms,0,blend_radius_m)
    |   movel([0.064703, -1.417356, -2.543784, -0.751249, 1.570796, 1.635499],accel_mss,speed_ms,0,blend_radius_m)
    |   movel([0.064470, -1.417487, -2.543684, -0.751218, 1.570796, 1.635266],accel_mss,speed_ms,0,blend_radius_m)
    |   movel([0.064153, -1.417621, -2.543582, -0.751186, 1.570796, 1.634949],accel_mss,speed_ms,0,blend_radius_m)
    |   movel([0.063688, -1.417783, -2.543459, -0.751147, 1.570796, 1.634484],accel_mss,speed_ms,0,blend_radius_m)
    |   movel([0.062952, -1.417996, -2.543297, -0.751096, 1.570796, 1.633749],accel_mss,speed_ms,0,blend_radius_m)
    |   movel([0.062645, -1.417969, -2.543318, -0.751102, 1.570796, 1.633441],accel_mss,speed_ms,0,blend_radius_m)
    |   movel([0.062507, -1.417741, -2.543491, -0.751157, 1.570796, 1.633304],accel_mss,speed_ms,0,blend_radius_m)
    |   movel([0.062499, -1.417093, -2.543983, -0.751312, 1.570796, 1.633295],accel_mss,speed_ms,0,blend_radius_m)
    |   movel([0.062527, -1.416327, -2.544565, -0.751497, 1.570796, 1.633324],accel_mss,speed_ms,0,blend_radius_m)
    |   speed_ms = 0.003
    |   movel([0.062527, -1.419519, -2.545993, -0.746877, 1.570796, 1.633324],accel_mss,speed_ms,0,blend_radius_m)
    |   speed_ms = 0.007
    |   movel([0.063795, -1.419220, -2.546221, -0.746948, 1.570796, 1.634591],accel_mss,speed_ms,0,blend_radius_m)
    |   movel([0.064285, -1.419107, -2.546307, -0.746975, 1.570796, 1.635081],accel_mss,speed_ms,0,blend_radius_m)
    |   movel([0.064715, -1.419015, -2.546377, -0.746997, 1.570796, 1.635511],accel_mss,speed_ms,0,blend_radius_m)
    |   movel([0.065077, -1.418941, -2.546433, -0.747014, 1.570796, 1.635874],accel_mss,speed_ms,0,blend_radius_m)
    |   movel([0.065199, -1.419130, -2.546290, -0.746969, 1.570796, 1.635995],accel_mss,speed_ms,0,blend_radius_m)
    |   movel([0.065192, -1.419550, -2.545970, -0.746869, 1.570796, 1.635988],accel_mss,speed_ms,0,blend_radius_m)
    |   movel([0.065156, -1.419861, -2.545732, -0.746795, 1.570796, 1.635953],accel_mss,speed_ms,0,blend_radius_m)
    |   movel([0.065014, -1.420241, -2.545442, -0.746705, 1.570796, 1.635811],accel_mss,speed_ms,0,blend_radius_m)
    |   movel([0.064703, -1.420545, -2.545210, -0.746633, 1.570796, 1.635499],accel_mss,speed_ms,0,blend_radius_m)
    |   movel([0.064470, -1.420676, -2.545110, -0.746603, 1.570796, 1.635266],accel_mss,speed_ms,0,blend_radius_m)
    |   movel([0.064153, -1.420810, -2.545008, -0.746571, 1.570796, 1.634949],accel_mss,speed_ms,0,blend_radius_m)
    |   movel([0.063688, -1.420971, -2.544885, -0.746533, 1.570796, 1.634484],accel_mss,speed_ms,0,blend_radius_m)
    |   movel([0.062952, -1.421183, -2.544723, -0.746483, 1.570796, 1.633749],accel_mss,speed_ms,0,blend_radius_m)
    |   movel([0.062645, -1.421157, -2.544743, -0.746489, 1.570796, 1.633441],accel_mss,speed_ms,0,blend_radius_m)
    |   movel([0.062507, -1.420930, -2.544916, -0.746543, 1.570796, 1.633304],accel_mss,speed_ms,0,blend_radius_m)
    |   movel([0.062499, -1.420284, -2.545410, -0.746695, 1.570796, 1.633295],accel_mss,speed_ms,0,blend_radius_m)
    |   movel([0.062527, -1.419519, -2.545993, -0.746877, 1.570796, 1.633324],accel_mss,speed_ms,0,blend_radius_m)
    |   speed_ms = 0.003
    |   movel([0.062527, -1.406871, -2.540231, -0.765286, 1.570796, 1.633324],accel_mss,speed_ms,0,blend_radius_m)
    |   speed_ms = 1.000
    |   movel([0.062527, -1.382550, -2.528315, -0.801524, 1.570796, 1.633324],accel_mss,speed_ms,0,blend_radius_m)
    |   movel([0.063592, -1.384530, -2.526885, -0.800974, 1.570796, 1.634388],accel_mss,speed_ms,0,blend_radius_m)
    |   movel([0.063592, -1.408813, -2.538777, -0.764799, 1.570796, 1.634388],accel_mss,speed_ms,0,blend_radius_m)
    |   speed_ms = 0.003
    |   movel([0.063592, -1.418253, -2.543102, -0.751035, 1.570796, 1.634388],accel_mss,speed_ms,0,blend_radius_m)
    |   speed_ms = 0.007
    |   movel([0.063854, -1.418154, -2.543177, -0.751058, 1.570796, 1.634651],accel_mss,speed_ms,0,blend_radius_m)
    |   movel([0.063749, -1.418375, -2.543008, -0.751005, 1.570796, 1.634545],accel_mss,speed_ms,0,blend_radius_m)
    |   movel([0.063517, -1.418344, -2.543032, -0.751013, 1.570796, 1.634313],accel_mss,speed_ms,0,blend_radius_m)
    |   speed_ms = 0.003
    |   movel([0.063592, -1.421440, -2.544527, -0.746423, 1.570796, 1.634388],accel_mss,speed_ms,0,blend_radius_m)
    |   speed_ms = 0.007
    |   movel([0.063854, -1.421342, -2.544602, -0.746446, 1.570796, 1.634651],accel_mss,speed_ms,0,blend_radius_m)
    |   movel([0.063749, -1.421562, -2.544433, -0.746394, 1.570796, 1.634545],accel_mss,speed_ms,0,blend_radius_m)
    |   movel([0.063517, -1.421531, -2.544457, -0.746401, 1.570796, 1.634313],accel_mss,speed_ms,0,blend_radius_m)
    |   speed_ms = 0.003
    |   movel([0.063592, -1.408813, -2.538777, -0.764799, 1.570796, 1.634388],accel_mss,speed_ms,0,blend_radius_m)
    |   speed_ms = 1.000
    |   movel([0.063592, -1.384530, -2.526885, -0.800974, 1.570796, 1.634388],accel_mss,speed_ms,0,blend_radius_m)
    |   movel([0.072778, -1.380851, -2.529537, -0.802001, 1.570796, 1.643574],accel_mss,speed_ms,0,blend_radius_m)
    |   movel([0.072778, -1.405204, -2.541475, -0.765709, 1.570796, 1.643574],accel_mss,speed_ms,0,blend_radius_m)
    |   speed_ms = 0.003
    |   movel([0.072778, -1.414673, -2.545817, -0.751899, 1.570796, 1.643574],accel_mss,speed_ms,0,blend_radius_m)
    |   speed_ms = 0.007
    |   movel([0.072754, -1.414237, -2.546146, -0.752005, 1.570796, 1.643550],accel_mss,speed_ms,0,blend_radius_m)
    |   movel([0.072827, -1.413744, -2.546519, -0.752126, 1.570796, 1.643623],accel_mss,speed_ms,0,blend_radius_m)
    |   movel([0.073001, -1.413335, -2.546827, -0.752227, 1.570796, 1.643797],accel_mss,speed_ms,0,blend_radius_m)
    |   movel([0.073524, -1.412666, -2.547331, -0.752392, 1.570796, 1.644320],accel_mss,speed_ms,0,blend_radius_m)
    |   movel([0.074243, -1.412069, -2.547781, -0.752540, 1.570796, 1.645040],accel_mss,speed_ms,0,blend_radius_m)
    |   movel([0.075186, -1.411533, -2.548183, -0.752673, 1.570796, 1.645983],accel_mss,speed_ms,0,blend_radius_m)
    |   movel([0.076383, -1.411042, -2.548552, -0.752795, 1.570796, 1.647179],accel_mss,speed_ms,0,blend_radius_m)
    |   movel([0.078821, -1.410334, -2.549083, -0.752972, 1.570796, 1.649617],accel_mss,speed_ms,0,blend_radius_m)
    |   movel([0.080585, -1.410209, -2.549177, -0.753003, 1.570796, 1.651381],accel_mss,speed_ms,0,blend_radius_m)
    |   movel([0.081607, -1.410656, -2.548842, -0.752891, 1.570796, 1.652403],accel_mss,speed_ms,0,blend_radius_m)
    |   movel([0.081913, -1.411602, -2.548132, -0.752655, 1.570796, 1.652709],accel_mss,speed_ms,0,blend_radius_m)
    |   movel([0.081873, -1.411895, -2.547911, -0.752583, 1.570796, 1.652669],accel_mss,speed_ms,0,blend_radius_m)
    |   movel([0.081731, -1.412271, -2.547629, -0.752489, 1.570796, 1.652528],accel_mss,speed_ms,0,blend_radius_m)
    |   movel([0.080649, -1.413002, -2.547079, -0.752309, 1.570796, 1.651445],accel_mss,speed_ms,0,blend_radius_m)
    |   movel([0.077230, -1.414010, -2.546318, -0.752061, 1.570796, 1.648026],accel_mss,speed_ms,0,blend_radius_m)
    |   movel([0.073822, -1.414927, -2.545625, -0.751837, 1.570796, 1.644619],accel_mss,speed_ms,0,blend_radius_m)
    |   movel([0.072922, -1.414873, -2.545666, -0.751850, 1.570796, 1.643719],accel_mss,speed_ms,0,blend_radius_m)
    |   movel([0.072778, -1.414673, -2.545817, -0.751899, 1.570796, 1.643574],accel_mss,speed_ms,0,blend_radius_m)
    |   speed_ms = 0.003
    |   movel([0.072778, -1.417870, -2.547248, -0.747271, 1.570796, 1.643574],accel_mss,speed_ms,0,blend_radius_m)
    |   speed_ms = 0.007
    |   movel([0.072754, -1.417436, -2.547578, -0.747375, 1.570796, 1.643550],accel_mss,speed_ms,0,blend_radius_m)
    |   movel([0.072827, -1.416944, -2.547951, -0.747494, 1.570796, 1.643623],accel_mss,speed_ms,0,blend_radius_m)
    |   movel([0.073001, -1.416536, -2.548260, -0.747593, 1.570796, 1.643797],accel_mss,speed_ms,0,blend_radius_m)
    |   movel([0.073524, -1.415869, -2.548765, -0.747755, 1.570796, 1.644320],accel_mss,speed_ms,0,blend_radius_m)
    |   movel([0.074243, -1.415273, -2.549216, -0.747900, 1.570796, 1.645040],accel_mss,speed_ms,0,blend_radius_m)
    |   movel([0.075186, -1.414739, -2.549619, -0.748031, 1.570796, 1.645983],accel_mss,speed_ms,0,blend_radius_m)
    |   movel([0.076383, -1.414250, -2.549988, -0.748151, 1.570796, 1.647179],accel_mss,speed_ms,0,blend_radius_m)
    |   movel([0.078821, -1.413544, -2.550521, -0.748325, 1.570796, 1.649617],accel_mss,speed_ms,0,blend_radius_m)
    |   movel([0.080585, -1.413419, -2.550614, -0.748356, 1.570796, 1.651381],accel_mss,speed_ms,0,blend_radius_m)
    |   movel([0.081607, -1.413864, -2.550279, -0.748246, 1.570796, 1.652403],accel_mss,speed_ms,0,blend_radius_m)
    |   movel([0.081913, -1.414808, -2.549567, -0.748014, 1.570796, 1.652709],accel_mss,speed_ms,0,blend_radius_m)
    |   movel([0.081873, -1.415100, -2.549346, -0.747942, 1.570796, 1.652669],accel_mss,speed_ms,0,blend_radius_m)
    |   movel([0.081731, -1.415475, -2.549063, -0.747851, 1.570796, 1.652528],accel_mss,speed_ms,0,blend_radius_m)
    |   movel([0.080649, -1.416204, -2.548512, -0.747674, 1.570796, 1.651445],accel_mss,speed_ms,0,blend_radius_m)
    |   movel([0.077230, -1.417209, -2.547750, -0.747430, 1.570796, 1.648026],accel_mss,speed_ms,0,blend_radius_m)
    |   movel([0.073822, -1.418123, -2.547056, -0.747210, 1.570796, 1.644619],accel_mss,speed_ms,0,blend_radius_m)
    |   movel([0.072922, -1.418070, -2.547096, -0.747223, 1.570796, 1.643719],accel_mss,speed_ms,0,blend_radius_m)
    |   movel([0.072778, -1.417870, -2.547248, -0.747271, 1.570796, 1.643574],accel_mss,speed_ms,0,blend_radius_m)
    |   speed_ms = 0.003
    |   movel([0.072778, -1.405204, -2.541475, -0.765709, 1.570796, 1.643574],accel_mss,speed_ms,0,blend_radius_m)
    |   speed_ms = 1.000
    |   movel([0.072778, -1.380851, -2.529537, -0.802001, 1.570796, 1.643574],accel_mss,speed_ms,0,blend_radius_m)
    |   movel([0.074421, -1.377304, -2.532077, -0.803009, 1.570796, 1.645217],accel_mss,speed_ms,0,blend_radius_m)
    |   movel([0.074421, -1.401724, -2.544059, -0.766606, 1.570796, 1.645217],accel_mss,speed_ms,0,blend_radius_m)
    |   speed_ms = 0.003
    |   movel([0.074421, -1.411221, -2.548417, -0.752750, 1.570796, 1.645217],accel_mss,speed_ms,0,blend_radius_m)
    |   speed_ms = 0.007
    |   movel([0.074165, -1.411024, -2.548565, -0.752799, 1.570796, 1.644961],accel_mss,speed_ms,0,blend_radius_m)
    |   movel([0.074354, -1.410618, -2.548870, -0.752901, 1.570796, 1.645150],accel_mss,speed_ms,0,blend_radius_m)
    |   movel([0.074666, -1.410362, -2.549062, -0.752965, 1.570796, 1.645462],accel_mss,speed_ms,0,blend_radius_m)
    |   movel([0.074969, -1.410185, -2.549195, -0.753009, 1.570796, 1.645765],accel_mss,speed_ms,0,blend_radius_m)
    |   movel([0.075423, -1.410001, -2.549333, -0.753055, 1.570796, 1.646220],accel_mss,speed_ms,0,blend_radius_m)
    |   movel([0.076121, -1.409766, -2.549509, -0.753114, 1.570796, 1.646917],accel_mss,speed_ms,0,blend_radius_m)
    |   movel([0.077322, -1.409397, -2.549785, -0.753207, 1.570796, 1.648119],accel_mss,speed_ms,0,blend_radius_m)
    |   movel([0.078883, -1.408949, -2.550119, -0.753320, 1.570796, 1.649680],accel_mss,speed_ms,0,blend_radius_m)
    |   movel([0.079928, -1.408708, -2.550300, -0.753381, 1.570796, 1.650725],accel_mss,speed_ms,0,blend_radius_m)
    |   movel([0.080636, -1.408620, -2.550365, -0.753403, 1.570796, 1.651433],accel_mss,speed_ms,0,blend_radius_m)
    |   movel([0.081039, -1.408696, -2.550309, -0.753384, 1.570796, 1.651835],accel_mss,speed_ms,0,blend_radius_m)
    |   movel([0.081219, -1.408932, -2.550132, -0.753324, 1.570796, 1.652015],accel_mss,speed_ms,0,blend_radius_m)
    |   movel([0.081009, -1.409281, -2.549872, -0.753237, 1.570796, 1.651806],accel_mss,speed_ms,0,blend_radius_m)
    |   movel([0.080717, -1.409508, -2.549702, -0.753179, 1.570796, 1.651513],accel_mss,speed_ms,0,blend_radius_m)
    |   movel([0.079948, -1.409576, -2.549651, -0.753162, 1.570796, 1.650744],accel_mss,speed_ms,0,blend_radius_m)
    |   movel([0.079003, -1.409713, -2.549549, -0.753128, 1.570796, 1.649800],accel_mss,speed_ms,0,blend_radius_m)
    |   movel([0.077590, -1.410075, -2.549277, -0.753037, 1.570796, 1.648387],accel_mss,speed_ms,0,blend_radius_m)
    |   movel([0.076171, -1.410515, -2.548947, -0.752926, 1.570796, 1.646967],accel_mss,speed_ms,0,blend_radius_m)
    |   movel([0.075220, -1.410915, -2.548648, -0.752827, 1.570796, 1.646016],accel_mss,speed_ms,0,blend_radius_m)
    |   movel([0.074765, -1.411137, -2.548481, -0.752771, 1.570796, 1.645561],accel_mss,speed_ms,0,blend_radius_m)
    |   movel([0.074421, -1.411221, -2.548417, -0.752750, 1.570796, 1.645217],accel_mss,speed_ms,0,blend_radius_m)
    |   speed_ms = 0.003
    |   movel([0.074421, -1.414429, -2.549853, -0.748107, 1.570796, 1.645217],accel_mss,speed_ms,0,blend_radius_m)
    |   speed_ms = 0.007
    |   movel([0.074165, -1.414232, -2.550002, -0.748155, 1.570796, 1.644961],accel_mss,speed_ms,0,blend_radius_m)
    |   movel([0.074354, -1.413827, -2.550307, -0.748255, 1.570796, 1.645150],accel_mss,speed_ms,0,blend_radius_m)
    |   movel([0.074666, -1.413572, -2.550499, -0.748318, 1.570796, 1.645462],accel_mss,speed_ms,0,blend_radius_m)
    |   movel([0.074969, -1.413395, -2.550632, -0.748361, 1.570796, 1.645765],accel_mss,speed_ms,0,blend_radius_m)
    |   movel([0.075423, -1.413212, -2.550771, -0.748407, 1.570796, 1.646220],accel_mss,speed_ms,0,blend_radius_m)
    |   movel([0.076121, -1.412977, -2.550947, -0.748465, 1.570796, 1.646917],accel_mss,speed_ms,0,blend_radius_m)
    |   movel([0.077322, -1.412609, -2.551224, -0.748556, 1.570796, 1.648119],accel_mss,speed_ms,0,blend_radius_m)
    |   movel([0.078883, -1.412163, -2.551559, -0.748667, 1.570796, 1.649680],accel_mss,speed_ms,0,blend_radius_m)
    |   movel([0.079928, -1.411922, -2.551740, -0.748727, 1.570796, 1.650725],accel_mss,speed_ms,0,blend_radius_m)
    |   movel([0.080636, -1.411835, -2.551805, -0.748749, 1.570796, 1.651433],accel_mss,speed_ms,0,blend_radius_m)
    |   movel([0.081039, -1.411910, -2.551749, -0.748730, 1.570796, 1.651835],accel_mss,speed_ms,0,blend_radius_m)
    |   movel([0.081219, -1.412146, -2.551572, -0.748671, 1.570796, 1.652015],accel_mss,speed_ms,0,blend_radius_m)
    |   movel([0.081009, -1.412493, -2.551311, -0.748585, 1.570796, 1.651806],accel_mss,speed_ms,0,blend_radius_m)
    |   movel([0.080717, -1.412720, -2.551141, -0.748529, 1.570796, 1.651513],accel_mss,speed_ms,0,blend_radius_m)
    |   movel([0.079948, -1.412788, -2.551089, -0.748512, 1.570796, 1.650744],accel_mss,speed_ms,0,blend_radius_m)
    |   movel([0.079003, -1.412924, -2.550987, -0.748478, 1.570796, 1.649800],accel_mss,speed_ms,0,blend_radius_m)
    |   movel([0.077590, -1.413286, -2.550715, -0.748388, 1.570796, 1.648387],accel_mss,speed_ms,0,blend_radius_m)
    |   movel([0.076171, -1.413724, -2.550384, -0.748280, 1.570796, 1.646967],accel_mss,speed_ms,0,blend_radius_m)
    |   movel([0.075220, -1.414123, -2.550084, -0.748182, 1.570796, 1.646016],accel_mss,speed_ms,0,blend_radius_m)
    |   movel([0.074765, -1.414344, -2.549917, -0.748128, 1.570796, 1.645561],accel_mss,speed_ms,0,blend_radius_m)
    |   movel([0.074421, -1.414429, -2.549853, -0.748107, 1.570796, 1.645217],accel_mss,speed_ms,0,blend_radius_m)
    |   speed_ms = 0.003
    |   movel([0.074421, -1.401724, -2.544059, -0.766606, 1.570796, 1.645217],accel_mss,speed_ms,0,blend_radius_m)
    |   speed_ms = 1.000
    |   movel([0.074421, -1.377304, -2.532077, -0.803009, 1.570796, 1.645217],accel_mss,speed_ms,0,blend_radius_m)
    |   movel([0.074736, -1.375712, -2.533211, -0.803467, 1.570796, 1.645532],accel_mss,speed_ms,0,blend_radius_m)
    |   movel([0.074736, -1.400162, -2.545213, -0.767014, 1.570796, 1.645532],accel_mss,speed_ms,0,blend_radius_m)
    |   speed_ms = 0.003
    |   movel([0.074736, -1.409672, -2.549579, -0.753138, 1.570796, 1.645532],accel_mss,speed_ms,0,blend_radius_m)
    |   speed_ms = 0.007
    |   movel([0.074490, -1.409676, -2.549576, -0.753137, 1.570796, 1.645287],accel_mss,speed_ms,0,blend_radius_m)
    |   movel([0.074368, -1.409543, -2.549675, -0.753170, 1.570796, 1.645164],accel_mss,speed_ms,0,blend_radius_m)
    |   movel([0.074367, -1.409330, -2.549835, -0.753224, 1.570796, 1.645164],accel_mss,speed_ms,0,blend_radius_m)
    |   movel([0.074493, -1.409079, -2.550022, -0.753287, 1.570796, 1.645290],accel_mss,speed_ms,0,blend_radius_m)
    |   movel([0.074719, -1.408846, -2.550197, -0.753346, 1.570796, 1.645515],accel_mss,speed_ms,0,blend_radius_m)
    |   movel([0.075001, -1.408669, -2.550329, -0.753391, 1.570796, 1.645798],accel_mss,speed_ms,0,blend_radius_m)
    |   movel([0.075428, -1.408490, -2.550463, -0.753436, 1.570796, 1.646224],accel_mss,speed_ms,0,blend_radius_m)
    |   movel([0.076116, -1.408259, -2.550635, -0.753495, 1.570796, 1.646913],accel_mss,speed_ms,0,blend_radius_m)
    |   movel([0.077432, -1.407859, -2.550934, -0.753597, 1.570796, 1.648228],accel_mss,speed_ms,0,blend_radius_m)
    |   movel([0.079178, -1.407349, -2.551313, -0.753726, 1.570796, 1.649974],accel_mss,speed_ms,0,blend_radius_m)
    |   movel([0.080115, -1.407122, -2.551483, -0.753784, 1.570796, 1.650912],accel_mss,speed_ms,0,blend_radius_m)
    |   movel([0.080700, -1.407049, -2.551537, -0.753803, 1.570796, 1.651497],accel_mss,speed_ms,0,blend_radius_m)
    |   movel([0.081098, -1.407114, -2.551489, -0.753786, 1.570796, 1.651894],accel_mss,speed_ms,0,blend_radius_m)
    |   movel([0.081299, -1.407228, -2.551404, -0.753757, 1.570796, 1.652096],accel_mss,speed_ms,0,blend_radius_m)
    |   movel([0.081309, -1.407519, -2.551187, -0.753683, 1.570796, 1.652105],accel_mss,speed_ms,0,blend_radius_m)
    |   movel([0.081126, -1.407734, -2.551027, -0.753628, 1.570796, 1.651922],accel_mss,speed_ms,0,blend_radius_m)
    |   movel([0.080817, -1.407938, -2.550875, -0.753576, 1.570796, 1.651613],accel_mss,speed_ms,0,blend_radius_m)
    |   movel([0.080255, -1.408044, -2.550795, -0.753549, 1.570796, 1.651051],accel_mss,speed_ms,0,blend_radius_m)
    |   movel([0.079381, -1.408214, -2.550669, -0.753506, 1.570796, 1.650177],accel_mss,speed_ms,0,blend_radius_m)
    |   movel([0.077678, -1.408681, -2.550320, -0.753388, 1.570796, 1.648474],accel_mss,speed_ms,0,blend_radius_m)
    |   movel([0.075967, -1.409187, -2.549942, -0.753260, 1.570796, 1.646764],accel_mss,speed_ms,0,blend_radius_m)
    |   movel([0.075186, -1.409493, -2.549713, -0.753183, 1.570796, 1.645982],accel_mss,speed_ms,0,blend_radius_m)
    |   movel([0.074925, -1.409608, -2.549627, -0.753154, 1.570796, 1.645722],accel_mss,speed_ms,0,blend_radius_m)
    |   speed_ms = 0.003
    |   movel([0.074736, -1.412884, -2.551017, -0.748488, 1.570796, 1.645532],accel_mss,speed_ms,0,blend_radius_m)
    |   speed_ms = 0.007
    |   movel([0.074490, -1.412888, -2.551014, -0.748487, 1.570796, 1.645287],accel_mss,speed_ms,0,blend_radius_m)
    |   movel([0.074368, -1.412755, -2.551114, -0.748520, 1.570796, 1.645164],accel_mss,speed_ms,0,blend_radius_m)
    |   movel([0.074367, -1.412543, -2.551274, -0.748572, 1.570796, 1.645164],accel_mss,speed_ms,0,blend_radius_m)
    |   movel([0.074493, -1.412293, -2.551462, -0.748635, 1.570796, 1.645290],accel_mss,speed_ms,0,blend_radius_m)
    |   movel([0.074719, -1.412060, -2.551637, -0.748693, 1.570796, 1.645515],accel_mss,speed_ms,0,blend_radius_m)
    |   movel([0.075001, -1.411883, -2.551769, -0.748737, 1.570796, 1.645798],accel_mss,speed_ms,0,blend_radius_m)
    |   movel([0.075428, -1.411705, -2.551903, -0.748781, 1.570796, 1.646224],accel_mss,speed_ms,0,blend_radius_m)
    |   movel([0.076116, -1.411474, -2.552076, -0.748839, 1.570796, 1.646913],accel_mss,speed_ms,0,blend_radius_m)
    |   movel([0.077432, -1.411075, -2.552375, -0.748938, 1.570796, 1.648228],accel_mss,speed_ms,0,blend_radius_m)
    |   movel([0.079178, -1.410568, -2.552756, -0.749066, 1.570796, 1.649974],accel_mss,speed_ms,0,blend_radius_m)
    |   movel([0.080115, -1.410341, -2.552926, -0.749123, 1.570796, 1.650912],accel_mss,speed_ms,0,blend_radius_m)
    |   movel([0.080700, -1.410268, -2.552980, -0.749141, 1.570796, 1.651497],accel_mss,speed_ms,0,blend_radius_m)
    |   movel([0.081098, -1.410332, -2.552932, -0.749125, 1.570796, 1.651894],accel_mss,speed_ms,0,blend_radius_m)
    |   movel([0.081299, -1.410446, -2.552846, -0.749096, 1.570796, 1.652096],accel_mss,speed_ms,0,blend_radius_m)
    |   movel([0.081309, -1.410737, -2.552629, -0.749023, 1.570796, 1.652105],accel_mss,speed_ms,0,blend_radius_m)
    |   movel([0.081126, -1.410951, -2.552468, -0.748970, 1.570796, 1.651922],accel_mss,speed_ms,0,blend_radius_m)
    |   movel([0.080817, -1.411154, -2.552316, -0.748919, 1.570796, 1.651613],accel_mss,speed_ms,0,blend_radius_m)
    |   movel([0.080255, -1.411261, -2.552236, -0.748892, 1.570796, 1.651051],accel_mss,speed_ms,0,blend_radius_m)
    |   movel([0.079381, -1.411429, -2.552110, -0.748850, 1.570796, 1.650177],accel_mss,speed_ms,0,blend_radius_m)
    |   movel([0.077678, -1.411896, -2.551760, -0.748733, 1.570796, 1.648474],accel_mss,speed_ms,0,blend_radius_m)
    |   movel([0.075967, -1.412400, -2.551381, -0.748608, 1.570796, 1.646764],accel_mss,speed_ms,0,blend_radius_m)
    |   movel([0.075186, -1.412705, -2.551152, -0.748532, 1.570796, 1.645982],accel_mss,speed_ms,0,blend_radius_m)
    |   movel([0.074925, -1.412820, -2.551066, -0.748504, 1.570796, 1.645722],accel_mss,speed_ms,0,blend_radius_m)
    |   speed_ms = 0.003
    |   movel([0.074736, -1.400162, -2.545213, -0.767014, 1.570796, 1.645532],accel_mss,speed_ms,0,blend_radius_m)
    |   speed_ms = 1.000
    |   movel([0.074736, -1.375712, -2.533211, -0.803467, 1.570796, 1.645532],accel_mss,speed_ms,0,blend_radius_m)
    |   movel([0.075139, -1.373952, -2.534460, -0.803977, 1.570796, 1.645936],accel_mss,speed_ms,0,blend_radius_m)
    |   movel([0.075139, -1.398436, -2.546485, -0.767469, 1.570796, 1.645936],accel_mss,speed_ms,0,blend_radius_m)
    |   speed_ms = 0.003
    |   movel([0.075139, -1.407960, -2.550859, -0.753571, 1.570796, 1.645936],accel_mss,speed_ms,0,blend_radius_m)
    |   speed_ms = 0.007
    |   movel([0.074668, -1.408057, -2.550786, -0.753546, 1.570796, 1.645464],accel_mss,speed_ms,0,blend_radius_m)
    |   movel([0.074481, -1.407978, -2.550845, -0.753566, 1.570796, 1.645278],accel_mss,speed_ms,0,blend_radius_m)
    |   movel([0.074467, -1.407741, -2.551022, -0.753627, 1.570796, 1.645263],accel_mss,speed_ms,0,blend_radius_m)
    |   movel([0.074692, -1.407404, -2.551273, -0.753712, 1.570796, 1.645489],accel_mss,speed_ms,0,blend_radius_m)
    |   movel([0.075140, -1.407096, -2.551502, -0.753791, 1.570796, 1.645937],accel_mss,speed_ms,0,blend_radius_m)
    |   movel([0.075912, -1.406763, -2.551750, -0.753876, 1.570796, 1.646708],accel_mss,speed_ms,0,blend_radius_m)
    |   movel([0.077256, -1.406314, -2.552084, -0.753991, 1.570796, 1.648052],accel_mss,speed_ms,0,blend_radius_m)
    |   movel([0.078806, -1.405855, -2.552425, -0.754109, 1.570796, 1.649603],accel_mss,speed_ms,0,blend_radius_m)
    |   movel([0.079979, -1.405582, -2.552628, -0.754179, 1.570796, 1.650775],accel_mss,speed_ms,0,blend_radius_m)
    |   movel([0.080824, -1.405467, -2.552713, -0.754209, 1.570796, 1.651621],accel_mss,speed_ms,0,blend_radius_m)
    |   movel([0.081268, -1.405549, -2.552652, -0.754188, 1.570796, 1.652064],accel_mss,speed_ms,0,blend_radius_m)
    |   movel([0.081447, -1.405680, -2.552555, -0.754154, 1.570796, 1.652243],accel_mss,speed_ms,0,blend_radius_m)
    |   movel([0.081473, -1.405951, -2.552354, -0.754084, 1.570796, 1.652269],accel_mss,speed_ms,0,blend_radius_m)
    |   movel([0.081179, -1.406214, -2.552158, -0.754017, 1.570796, 1.651975],accel_mss,speed_ms,0,blend_radius_m)
    |   movel([0.080823, -1.406331, -2.552072, -0.753987, 1.570796, 1.651619],accel_mss,speed_ms,0,blend_radius_m)
    |   movel([0.080297, -1.406474, -2.551965, -0.753950, 1.570796, 1.651093],accel_mss,speed_ms,0,blend_radius_m)
    |   movel([0.079504, -1.406660, -2.551826, -0.753902, 1.570796, 1.650301],accel_mss,speed_ms,0,blend_radius_m)
